Yaskawa INFORM job: aprem2TRJ3.JBI

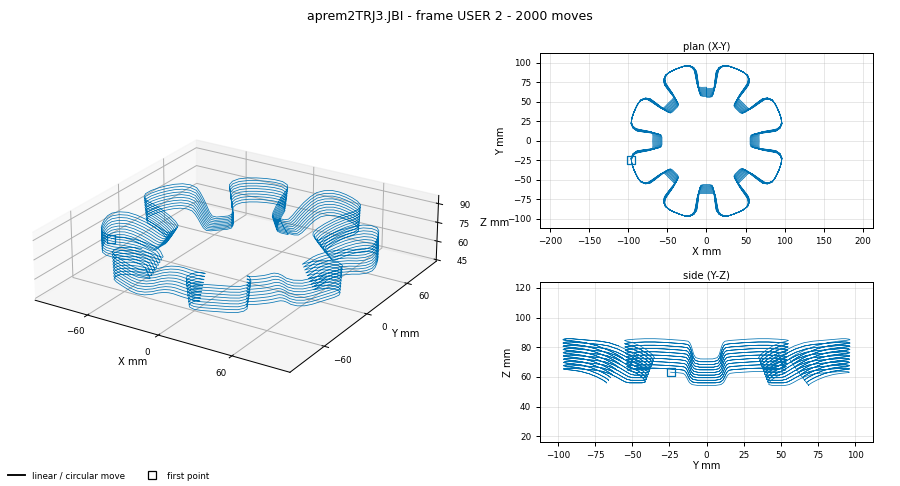
[picture p0: tool path of aprem2TRJ3.JBI in frame USER 2, 2000 of 2000 moves have a stored position in this frame; points joined in program order, loops and branches not executed]
/JOB
//NAME aprem2TRJ3
//POS
///NPOS 2000,0,2000,0,0,0
///USER 2
///TOOL 1
///POSTYPE USER
///RECTAN
///RCONF 1,0,0,0,0,0,0,0,0,0,0,0,0,0,0,0,0,0,0,0,0,0,0,0
C00000=-96.154,-24.159,63.210,179.7472,-2.4641,0.0000
C00001=-94.423,-19.246,62.877,177.2942,-4.1530,0.0000
C00002=-90.636,-15.942,62.469,172.7045,-3.4321,0.0000
C00003=-85.405,-14.621,61.698,172.2425,-1.7901,0.0000
C00004=-79.780,-13.569,60.151,174.0266,-1.3203,0.0000
C00005=-74.809,-12.586,58.158,176.9961,-0.7607,0.0000
C00006=-71.127,-11.507,56.252,-176.5790,1.2623,0.0000
C00007=-69.044,-9.699,54.888,-163.7838,26.3525,0.0000
C00008=-68.619,-6.200,54.350,-178.9508,38.3093,0.0000
C00009=-68.781,-2.945,54.326,177.7405,38.7530,0.0000
C00010=-68.843,0.000,54.342,179.9996,38.7765,0.0000
C00011=-68.781,2.945,54.326,-177.7401,38.7530,0.0000
C00012=-68.619,6.200,54.350,178.9482,38.3089,0.0000
C00013=-69.044,9.699,54.888,163.7840,26.3528,0.0000
C00014=-71.127,11.507,56.252,176.5790,1.2623,0.0000
C00015=-74.809,12.586,58.158,-176.9961,-0.7607,0.0000
C00016=-79.780,13.569,60.151,-174.0266,-1.3203,0.0000
C00017=-85.405,14.621,61.698,-172.2425,-1.7901,0.0000
C00018=-90.636,15.942,62.469,-172.7045,-3.4321,0.0000
C00019=-94.423,19.246,62.877,-177.2942,-4.1530,0.0000
C00020=-96.154,24.159,63.210,-179.7472,-2.4641,0.0000
C00021=-95.429,29.718,63.547,179.9546,-0.1514,0.0000
C00022=-93.512,35.416,63.770,179.9933,-0.0179,0.0000
C00023=-91.166,41.080,63.770,179.9921,-0.0174,0.0000
C00024=-88.493,46.465,63.547,179.9251,-0.1391,0.0000
C00025=-85.074,50.908,63.210,178.0786,-1.5643,0.0000
C00026=-80.376,53.158,62.877,175.1551,-1.0270,0.0000
C00027=-75.362,52.817,62.469,172.4279,2.7549,0.0000
C00028=-70.729,50.052,61.698,173.2462,4.2451,0.0000
C00029=-66.007,46.818,60.151,174.8410,3.3018,0.0000
C00030=-61.798,43.998,58.158,177.3380,1.5877,0.0000
C00031=-58.431,42.158,56.252,-176.6891,-1.5289,0.0000
C00032=-55.679,41.963,54.888,-150.9290,8.2296,0.0000
C00033=-52.905,44.137,54.350,-150.2488,28.6202,0.0000
C00034=-50.718,46.553,54.326,-151.6454,30.7727,0.0000
C00035=-48.679,48.679,54.342,-150.4014,29.5989,0.0000
C00036=-46.553,50.718,54.326,-149.2271,28.3544,0.0000
C00037=-44.137,52.905,54.350,-151.3816,29.7523,0.0000
C00038=-41.963,55.680,54.888,-171.7700,29.0711,0.0000
C00039=-42.158,58.431,56.252,178.4711,3.3109,0.0000
C00040=-43.998,61.798,58.158,-178.4123,-2.6620,0.0000
C00041=-46.818,66.007,60.151,-176.6982,-5.1590,0.0000
C00042=-50.052,70.729,61.698,-175.7549,-6.7538,0.0000
C00043=-52.817,75.362,62.469,-177.2451,-7.5721,0.0000
C00044=-53.158,80.376,62.877,178.9730,-4.8449,0.0000
C00045=-50.908,85.074,63.210,178.4357,-1.9214,0.0000
C00046=-46.465,88.493,63.547,179.8609,-0.0749,0.0000
C00047=-41.080,91.166,63.770,179.9826,-0.0079,0.0000
C00048=-35.416,93.512,63.770,179.9821,-0.0067,0.0000
C00049=-29.718,95.429,63.547,179.8486,-0.0454,0.0000
C00050=-24.159,96.154,63.210,177.5359,0.2528,0.0000
C00051=-19.246,94.423,62.877,175.8470,2.7058,0.0000
C00052=-15.942,90.636,62.469,176.5679,7.2955,0.0000
C00053=-14.621,85.405,61.698,178.2099,7.7575,0.0000
C00054=-13.569,79.780,60.151,178.6797,5.9734,0.0000
C00055=-12.586,74.809,58.158,179.2393,3.0039,0.0000
C00056=-11.507,71.127,56.252,-178.7377,-3.4210,0.0000
C00057=-9.699,69.044,54.888,-153.6472,-16.2160,0.0000
C00058=-6.200,68.619,54.350,-141.6911,-1.0518,0.0000
C00059=-2.945,68.781,54.326,-141.2470,2.2599,0.0000
C00060=0.000,68.843,54.342,-141.2235,-0.0004,0.0000
C00061=0.000,67.469,56.061,-141.5412,-0.0004,0.0000
C00062=2.820,67.413,56.044,-141.5636,-2.1988,0.0000
C00063=5.989,67.263,56.069,-142.0566,1.4090,0.0000
C00064=9.441,67.734,56.637,-154.9636,16.3668,0.0000
C00065=11.191,69.937,58.076,-179.1454,2.5065,0.0000
C00066=12.227,73.809,60.085,179.1943,-3.3815,0.0000
C00067=13.183,79.025,62.181,178.7261,-6.0865,0.0000
C00068=14.211,84.918,63.804,178.3204,-7.7435,0.0000
C00069=15.500,90.396,64.610,176.7328,-7.3164,0.0000
C00070=18.832,94.373,65.037,175.8897,-2.7823,0.0000
C00071=23.832,96.213,65.385,177.5484,-0.2740,0.0000
C00072=29.513,95.497,65.736,179.8479,0.0454,0.0000
C00073=35.347,93.539,65.969,179.9821,0.0067,0.0000
C00074=41.148,91.136,65.969,179.9826,0.0079,0.0000
C00075=46.658,88.395,65.736,179.8603,0.0754,0.0000
C00076=51.181,84.885,65.385,178.4595,1.9277,0.0000
C00077=53.416,80.048,65.037,179.0575,4.8686,0.0000
C00078=52.959,74.880,64.610,-177.1134,7.4719,0.0000
C00079=49.997,70.095,63.804,-175.6871,6.6669,0.0000
C00080=46.557,65.200,62.181,-176.5849,5.2066,0.0000
C00081=43.545,60.837,60.085,-178.1765,2.9610,0.0000
C00082=41.540,57.367,58.076,178.8310,-2.3765,0.0000
C00083=41.220,54.571,56.637,-173.0100,-28.2777,0.0000
C00084=43.327,51.796,56.069,-151.9006,-29.6278,0.0000
C00085=45.674,49.662,56.044,-149.5306,-28.1035,0.0000
C00086=47.708,47.708,56.061,-150.6800,-29.3196,0.0000
C00087=49.662,45.674,56.044,-151.8968,-30.4697,0.0000
C00088=51.797,43.327,56.069,-150.3712,-28.0975,0.0000
C00089=54.571,41.220,56.637,-151.7222,-6.9903,0.0000
C00090=57.367,41.540,58.076,-177.6235,1.1690,0.0000
C00091=60.837,43.545,60.085,177.0390,-1.8235,0.0000
C00092=65.200,46.557,62.181,174.7934,-3.4151,0.0000
C00093=70.095,49.997,63.804,173.3331,-4.3129,0.0000
C00094=74.880,52.959,64.610,172.5281,-2.8866,0.0000
C00095=80.048,53.416,65.037,175.1314,0.9425,0.0000
C00096=84.885,51.181,65.385,178.0723,1.5405,0.0000
C00097=88.395,46.658,65.736,179.9246,0.1397,0.0000
C00098=91.136,41.148,65.969,179.9921,0.0174,0.0000
C00099=93.539,35.347,65.969,179.9933,0.0179,0.0000
C00100=95.497,29.513,65.736,179.9546,0.1521,0.0000
C00101=96.213,23.832,65.385,-179.7260,2.4516,0.0000
C00102=94.373,18.832,65.037,-177.2177,4.1103,0.0000
C00103=90.396,15.500,64.610,-172.6836,3.2672,0.0000
C00104=84.918,14.211,63.804,-172.2565,1.6796,0.0000
C00105=79.025,13.183,62.181,-173.9135,1.2739,0.0000
C00106=73.809,12.227,60.085,-176.6185,0.8057,0.0000
C00107=69.937,11.191,58.076,177.4935,-0.8546,0.0000
C00108=67.734,9.441,56.637,163.6332,-25.0364,0.0000
C00109=67.263,5.989,56.069,178.5910,-37.9434,0.0000
C00110=67.413,2.820,56.044,-177.8012,-38.4364,0.0000
C00111=67.469,0.000,56.061,-179.9996,-38.4588,0.0000
C00112=67.413,-2.820,56.044,177.8008,-38.4364,0.0000
C00113=67.263,-5.989,56.069,-178.5883,-37.9429,0.0000
C00114=67.734,-9.441,56.637,-163.6333,-25.0366,0.0000
C00115=69.937,-11.191,58.076,-177.4935,-0.8546,0.0000
C00116=73.809,-12.227,60.085,176.6185,0.8057,0.0000
C00117=79.025,-13.183,62.181,173.9135,1.2739,0.0000
C00118=84.918,-14.211,63.804,172.2565,1.6796,0.0000
C00119=90.396,-15.500,64.610,172.6836,3.2672,0.0000
C00120=94.373,-18.832,65.037,177.2177,4.1103,0.0000
C00121=96.213,-23.832,65.385,179.7260,2.4516,0.0000
C00122=95.497,-29.513,65.736,-179.9546,0.1521,0.0000
C00123=93.539,-35.347,65.969,-179.9933,0.0179,0.0000
C00124=91.136,-41.148,65.969,-179.9921,0.0174,0.0000
C00125=88.395,-46.658,65.736,-179.9246,0.1397,0.0000
C00126=84.885,-51.181,65.385,-178.0723,1.5405,0.0000
C00127=80.048,-53.416,65.037,-175.1314,0.9425,0.0000
C00128=74.880,-52.959,64.610,-172.5281,-2.8866,0.0000
C00129=70.095,-49.997,63.804,-173.3331,-4.3129,0.0000
C00130=65.200,-46.557,62.181,-174.7934,-3.4151,0.0000
C00131=60.837,-43.545,60.085,-177.0390,-1.8235,0.0000
C00132=57.367,-41.540,58.076,177.6235,1.1690,0.0000
C00133=54.571,-41.220,56.637,151.7223,-6.9900,0.0000
C00134=51.796,-43.327,56.069,150.3722,-28.0994,0.0000
C00135=49.662,-45.674,56.044,151.8965,-30.4694,0.0000
C00136=47.708,-47.708,56.061,150.6804,-29.3200,0.0000
C00137=45.674,-49.662,56.044,149.5303,-28.1032,0.0000
C00138=43.327,-51.797,56.069,151.9025,-29.6288,0.0000
C00139=41.220,-54.571,56.637,173.0097,-28.2778,0.0000
C00140=41.540,-57.367,58.076,-178.8310,-2.3765,0.0000
C00141=43.545,-60.837,60.085,178.1765,2.9610,0.0000
C00142=46.557,-65.200,62.181,176.5849,5.2066,0.0000
C00143=49.997,-70.095,63.804,175.6871,6.6669,0.0000
C00144=52.959,-74.880,64.610,177.1134,7.4719,0.0000
C00145=53.416,-80.048,65.037,-179.0575,4.8686,0.0000
C00146=51.181,-84.885,65.385,-178.4595,1.9277,0.0000
C00147=46.658,-88.395,65.736,-179.8603,0.0754,0.0000
C00148=41.148,-91.136,65.969,-179.9826,0.0079,0.0000
C00149=35.347,-93.539,65.969,-179.9821,0.0067,0.0000
C00150=29.513,-95.497,65.736,-179.8479,0.0454,0.0000
C00151=23.832,-96.213,65.385,-177.5484,-0.2740,0.0000
C00152=18.832,-94.373,65.037,-175.8897,-2.7823,0.0000
C00153=15.500,-90.396,64.610,-176.7328,-7.3164,0.0000
C00154=14.211,-84.918,63.804,-178.3204,-7.7435,0.0000
C00155=13.183,-79.025,62.181,-178.7261,-6.0865,0.0000
C00156=12.227,-73.809,60.085,-179.1943,-3.3815,0.0000
C00157=11.191,-69.937,58.076,179.1454,2.5065,0.0000
C00158=9.441,-67.734,56.637,154.9636,16.3668,0.0000
C00159=5.989,-67.263,56.069,142.0566,1.4090,0.0000
C00160=2.820,-67.413,56.044,141.5636,-2.1988,0.0000
C00161=0.000,-67.469,56.061,141.5412,-0.0004,0.0000
C00162=0.000,-67.469,56.061,141.5412,-0.0004,0.0000
C00163=-2.820,-67.413,56.044,141.5636,2.1992,0.0000
C00164=-5.989,-67.263,56.069,142.0571,-1.4117,0.0000
C00165=-9.441,-67.734,56.637,154.9634,-16.3667,0.0000
C00166=-11.191,-69.937,58.076,179.1454,-2.5065,0.0000
C00167=-12.227,-73.809,60.085,-179.1943,3.3815,0.0000
C00168=-13.183,-79.025,62.181,-178.7261,6.0865,0.0000
C00169=-14.211,-84.918,63.804,-178.3204,7.7435,0.0000
C00170=-15.500,-90.396,64.610,-176.7328,7.3164,0.0000
C00171=-18.832,-94.373,65.037,-175.8897,2.7823,0.0000
C00172=-23.832,-96.213,65.385,-177.5484,0.2740,0.0000
C00173=-29.513,-95.497,65.736,-179.8479,-0.0454,0.0000
C00174=-35.347,-93.539,65.969,-179.9821,-0.0067,0.0000
C00175=-41.148,-91.136,65.969,-179.9826,-0.0079,0.0000
C00176=-46.658,-88.395,65.736,-179.8603,-0.0754,0.0000
C00177=-51.181,-84.885,65.385,-178.4595,-1.9277,0.0000
C00178=-53.416,-80.048,65.037,-179.0575,-4.8686,0.0000
C00179=-52.959,-74.880,64.610,177.1134,-7.4719,0.0000
C00180=-49.997,-70.095,63.804,175.6871,-6.6669,0.0000
C00181=-46.557,-65.200,62.181,176.5849,-5.2066,0.0000
C00182=-43.545,-60.837,60.085,178.1765,-2.9610,0.0000
C00183=-41.540,-57.367,58.076,-178.8310,2.3765,0.0000
C00184=-41.220,-54.571,56.637,173.0100,28.2777,0.0000
C00185=-43.327,-51.796,56.069,151.9006,29.6278,0.0000
C00186=-45.674,-49.662,56.044,149.5306,28.1035,0.0000
C00187=-47.708,-47.708,56.061,150.6800,29.3196,0.0000
C00188=-49.662,-45.674,56.044,151.8968,30.4697,0.0000
C00189=-51.797,-43.327,56.069,150.3712,28.0975,0.0000
C00190=-54.571,-41.220,56.637,151.7222,6.9903,0.0000
C00191=-57.367,-41.540,58.076,177.6235,-1.1690,0.0000
C00192=-60.837,-43.545,60.085,-177.0390,1.8235,0.0000
C00193=-65.200,-46.557,62.181,-174.7934,3.4151,0.0000
C00194=-70.095,-49.997,63.804,-173.3331,4.3129,0.0000
C00195=-74.880,-52.959,64.610,-172.5281,2.8866,0.0000
C00196=-80.048,-53.416,65.037,-175.1314,-0.9425,0.0000
C00197=-84.885,-51.181,65.385,-178.0723,-1.5405,0.0000
C00198=-88.395,-46.658,65.736,-179.9246,-0.1397,0.0000
C00199=-91.136,-41.148,65.969,-179.9921,-0.0174,0.0000
C00200=-93.539,-35.347,65.969,-179.9933,-0.0179,0.0000
C00201=-95.497,-29.513,65.736,-179.9546,-0.1521,0.0000
C00202=-96.213,-23.832,65.385,179.7260,-2.4516,0.0000
C00203=-94.373,-18.832,65.037,177.2177,-4.1103,0.0000
C00204=-90.396,-15.500,64.610,172.6836,-3.2672,0.0000
C00205=-84.918,-14.211,63.804,172.2565,-1.6796,0.0000
C00206=-79.025,-13.183,62.181,173.9135,-1.2739,0.0000
C00207=-73.809,-12.227,60.085,176.6185,-0.8057,0.0000
C00208=-69.937,-11.191,58.076,-177.4935,0.8546,0.0000
C00209=-67.734,-9.441,56.637,-163.6332,25.0364,0.0000
C00210=-67.263,-5.989,56.069,-178.5910,37.9434,0.0000
C00211=-67.413,-2.820,56.044,177.8012,38.4364,0.0000
C00212=-67.469,0.000,56.061,179.9996,38.4588,0.0000
C00213=-67.413,2.820,56.044,-177.8008,38.4364,0.0000
C00214=-67.263,5.989,56.069,178.5883,37.9429,0.0000
C00215=-67.734,9.441,56.637,163.6333,25.0366,0.0000
C00216=-69.937,11.191,58.076,177.4935,0.8546,0.0000
C00217=-73.809,12.227,60.085,-176.6185,-0.8057,0.0000
C00218=-79.025,13.183,62.181,-173.9135,-1.2739,0.0000
C00219=-84.918,14.211,63.804,-172.2565,-1.6796,0.0000
C00220=-90.396,15.500,64.610,-172.6836,-3.2672,0.0000
C00221=-94.373,18.832,65.037,-177.2177,-4.1103,0.0000
C00222=-96.213,23.832,65.385,-179.7260,-2.4516,0.0000
C00223=-95.497,29.513,65.736,179.9546,-0.1521,0.0000
C00224=-93.539,35.347,65.969,179.9933,-0.0179,0.0000
C00225=-91.136,41.148,65.969,179.9921,-0.0174,0.0000
C00226=-88.395,46.658,65.736,179.9246,-0.1397,0.0000
C00227=-84.885,51.181,65.385,178.0723,-1.5405,0.0000
C00228=-80.048,53.416,65.037,175.1314,-0.9425,0.0000
C00229=-74.880,52.959,64.610,172.5281,2.8866,0.0000
C00230=-70.095,49.997,63.804,173.3331,4.3129,0.0000
C00231=-65.200,46.557,62.181,174.7934,3.4151,0.0000
C00232=-60.837,43.545,60.085,177.0390,1.8235,0.0000
C00233=-57.367,41.540,58.076,-177.6235,-1.1690,0.0000
C00234=-54.571,41.220,56.637,-151.7223,6.9900,0.0000
C00235=-51.796,43.327,56.069,-150.3722,28.0994,0.0000
C00236=-49.662,45.674,56.044,-151.8965,30.4694,0.0000
C00237=-47.708,47.708,56.061,-150.6804,29.3200,0.0000
C00238=-45.674,49.662,56.044,-149.5303,28.1032,0.0000
C00239=-43.327,51.797,56.069,-151.9025,29.6288,0.0000
C00240=-41.220,54.571,56.637,-173.0097,28.2778,0.0000
C00241=-41.540,57.367,58.076,178.8310,2.3765,0.0000
C00242=-43.545,60.837,60.085,-178.1765,-2.9610,0.0000
C00243=-46.557,65.200,62.181,-176.5849,-5.2066,0.0000
C00244=-49.997,70.095,63.804,-175.6871,-6.6669,0.0000
C00245=-52.959,74.880,64.610,-177.1134,-7.4719,0.0000
C00246=-53.416,80.048,65.037,179.0575,-4.8686,0.0000
C00247=-51.181,84.885,65.385,178.4595,-1.9277,0.0000
C00248=-46.658,88.395,65.736,179.8603,-0.0754,0.0000
C00249=-41.148,91.136,65.969,179.9826,-0.0079,0.0000
C00250=-35.347,93.539,65.969,179.9821,-0.0067,0.0000
C00251=-29.513,95.497,65.736,179.8479,-0.0454,0.0000
C00252=-23.832,96.213,65.385,177.5484,0.2740,0.0000
C00253=-18.832,94.373,65.037,175.8897,2.7823,0.0000
C00254=-15.500,90.396,64.610,176.7328,7.3164,0.0000
C00255=-14.211,84.918,63.804,178.3204,7.7435,0.0000
C00256=-13.183,79.025,62.181,178.7261,6.0865,0.0000
C00257=-12.227,73.809,60.085,179.1943,3.3815,0.0000
C00258=-11.191,69.937,58.076,-179.1454,-2.5065,0.0000
C00259=-9.441,67.734,56.637,-154.9634,-16.3667,0.0000
C00260=-5.989,67.263,56.069,-142.0571,-1.4117,0.0000
C00261=-2.820,67.413,56.044,-141.5636,2.1992,0.0000
C00262=0.000,67.469,56.061,-141.5412,-0.0004,0.0000
C00263=0.000,66.107,57.788,-141.9405,-0.0005,0.0000
C00264=2.695,66.055,57.771,-141.9617,-2.1301,0.0000
C00265=5.779,65.917,57.797,-142.5088,1.7632,0.0000
C00266=9.185,66.436,58.394,-156.3340,16.3865,0.0000
C00267=10.880,68.762,59.909,-179.4729,1.6691,0.0000
C00268=11.874,72.826,62.021,179.1708,-3.6886,0.0000
C00269=12.805,78.288,64.219,178.7806,-6.1350,0.0000
C00270=13.814,84.445,65.915,178.4333,-7.6593,0.0000
C00271=15.073,90.163,66.756,176.9116,-7.2599,0.0000
C00272=18.432,94.325,67.200,175.9710,-2.8231,0.0000
C00273=23.517,96.271,67.561,177.5835,-0.2906,0.0000
C00274=29.315,95.562,67.927,179.8488,0.0450,0.0000
C00275=35.280,93.564,68.167,179.9823,0.0066,0.0000
C00276=41.213,91.107,68.167,179.9828,0.0078,0.0000
C00277=46.844,88.301,67.927,179.8613,0.0751,0.0000
C00278=51.445,84.703,67.561,178.4961,1.9145,0.0000
C00279=53.664,79.731,67.200,179.1443,4.8399,0.0000
C00280=53.097,74.413,66.756,-177.0274,7.3072,0.0000
C00281=49.944,69.479,65.915,-175.6680,6.5281,0.0000
C00282=46.303,64.413,64.219,-176.5119,5.2027,0.0000
C00283=43.100,59.892,62.021,-177.9754,3.1949,0.0000
C00284=40.929,56.315,59.909,179.1922,-1.5529,0.0000
C00285=40.483,53.472,58.394,-174.1779,-27.3765,0.0000
C00286=42.524,50.697,57.797,-152.4966,-29.4307,0.0000
C00287=44.802,48.614,57.771,-149.9071,-27.7853,0.0000
C00288=46.745,46.745,57.788,-151.0292,-28.9702,0.0000
C00289=48.613,44.802,57.771,-152.2149,-30.0932,0.0000
C00290=50.697,42.524,57.797,-150.5682,-27.5015,0.0000
C00291=53.472,40.483,58.395,-152.6235,-5.8223,0.0000
C00292=56.315,40.929,59.909,-178.4471,0.8078,0.0000
C00293=59.892,43.100,62.021,176.8051,-2.0246,0.0000
C00294=64.413,46.303,64.219,174.7973,-3.4881,0.0000
C00295=69.479,49.944,65.915,173.4719,-4.3320,0.0000
C00296=74.413,53.097,66.756,172.6928,-2.9726,0.0000
C00297=79.731,53.664,67.200,175.1601,0.8557,0.0000
C00298=84.703,51.445,67.561,178.0855,1.5039,0.0000
C00299=88.301,46.844,67.927,179.9249,0.1387,0.0000
C00300=91.107,41.213,68.167,179.9922,0.0172,0.0000
C00301=93.564,35.280,68.167,179.9934,0.0177,0.0000
C00302=95.562,29.315,67.927,179.9550,0.1512,0.0000
C00303=96.271,23.517,67.561,-179.7094,2.4165,0.0000
C00304=94.325,18.432,67.200,-177.1769,4.0290,0.0000
C00305=90.163,15.073,66.756,-172.7401,3.0884,0.0000
C00306=84.445,13.814,65.915,-172.3407,1.5667,0.0000
C00307=78.288,12.805,64.219,-173.8650,1.2194,0.0000
C00308=72.826,11.874,62.021,-176.3114,0.8292,0.0000
C00309=68.762,10.880,59.909,178.3309,-0.5271,0.0000
C00310=66.436,9.185,58.394,163.6135,-23.6660,0.0000
C00311=65.917,5.779,57.797,178.2368,-37.4912,0.0000
C00312=66.055,2.695,57.771,-177.8699,-38.0383,0.0000
C00313=66.107,0.000,57.788,-179.9995,-38.0595,0.0000
C00314=66.055,-2.695,57.771,177.8693,-38.0383,0.0000
C00315=65.917,-5.780,57.797,-178.2340,-37.4907,0.0000
C00316=66.436,-9.185,58.395,-163.6136,-23.6662,0.0000
C00317=68.762,-10.880,59.909,-178.3309,-0.5271,0.0000
C00318=72.826,-11.874,62.021,176.3114,0.8292,0.0000
C00319=78.288,-12.805,64.219,173.8650,1.2194,0.0000
C00320=84.445,-13.814,65.915,172.3407,1.5667,0.0000
C00321=90.163,-15.073,66.756,172.7401,3.0884,0.0000
C00322=94.325,-18.432,67.200,177.1769,4.0290,0.0000
C00323=96.271,-23.517,67.561,179.7094,2.4165,0.0000
C00324=95.562,-29.315,67.927,-179.9550,0.1512,0.0000
C00325=93.564,-35.280,68.167,-179.9934,0.0177,0.0000
C00326=91.107,-41.213,68.167,-179.9922,0.0172,0.0000
C00327=88.301,-46.844,67.927,-179.9249,0.1387,0.0000
C00328=84.703,-51.445,67.561,-178.0855,1.5039,0.0000
C00329=79.731,-53.664,67.200,-175.1601,0.8557,0.0000
C00330=74.413,-53.097,66.756,-172.6928,-2.9726,0.0000
C00331=69.479,-49.944,65.915,-173.4719,-4.3320,0.0000
C00332=64.413,-46.303,64.219,-174.7973,-3.4881,0.0000
C00333=59.892,-43.100,62.021,-176.8051,-2.0246,0.0000
C00334=56.315,-40.929,59.909,178.4471,0.8078,0.0000
C00335=53.472,-40.483,58.394,152.6235,-5.8221,0.0000
C00336=50.697,-42.524,57.797,150.5693,-27.5034,0.0000
C00337=48.614,-44.802,57.771,152.2147,-30.0929,0.0000
C00338=46.745,-46.745,57.788,151.0298,-28.9708,0.0000
C00339=44.802,-48.613,57.771,149.9068,-27.7851,0.0000
C00340=42.524,-50.697,57.797,152.4985,-29.4318,0.0000
C00341=40.483,-53.472,58.395,174.1777,-27.3765,0.0000
C00342=40.929,-56.315,59.909,-179.1922,-1.5529,0.0000
C00343=43.100,-59.892,62.021,177.9754,3.1949,0.0000
C00344=46.303,-64.413,64.219,176.5119,5.2027,0.0000
C00345=49.944,-69.479,65.915,175.6680,6.5281,0.0000
C00346=53.097,-74.413,66.756,177.0274,7.3072,0.0000
C00347=53.664,-79.731,67.200,-179.1443,4.8399,0.0000
C00348=51.445,-84.703,67.561,-178.4961,1.9145,0.0000
C00349=46.844,-88.301,67.927,-179.8613,0.0751,0.0000
C00350=41.213,-91.107,68.167,-179.9828,0.0078,0.0000
C00351=35.280,-93.564,68.167,-179.9823,0.0066,0.0000
C00352=29.315,-95.562,67.927,-179.8488,0.0450,0.0000
C00353=23.517,-96.271,67.561,-177.5835,-0.2906,0.0000
C00354=18.432,-94.325,67.200,-175.9710,-2.8231,0.0000
C00355=15.073,-90.163,66.756,-176.9116,-7.2599,0.0000
C00356=13.814,-84.445,65.915,-178.4333,-7.6593,0.0000
C00357=12.805,-78.288,64.219,-178.7806,-6.1350,0.0000
C00358=11.874,-72.826,62.021,-179.1708,-3.6886,0.0000
C00359=10.880,-68.762,59.909,179.4729,1.6691,0.0000
C00360=9.185,-66.436,58.394,156.3340,16.3865,0.0000
C00361=5.779,-65.917,57.797,142.5088,1.7632,0.0000
C00362=2.695,-66.055,57.771,141.9617,-2.1301,0.0000
C00363=0.000,-66.107,57.788,141.9405,-0.0005,0.0000
C00364=0.000,-66.107,57.788,141.9405,-0.0005,0.0000
C00365=-2.695,-66.055,57.771,141.9617,2.1307,0.0000
C00366=-5.780,-65.917,57.797,142.5093,-1.7660,0.0000
C00367=-9.185,-66.436,58.395,156.3338,-16.3864,0.0000
C00368=-10.880,-68.762,59.909,179.4729,-1.6691,0.0000
C00369=-11.874,-72.826,62.021,-179.1708,3.6886,0.0000
C00370=-12.805,-78.288,64.219,-178.7806,6.1350,0.0000
C00371=-13.814,-84.445,65.915,-178.4333,7.6593,0.0000
C00372=-15.073,-90.163,66.756,-176.9116,7.2599,0.0000
C00373=-18.432,-94.325,67.200,-175.9710,2.8231,0.0000
C00374=-23.517,-96.271,67.561,-177.5835,0.2906,0.0000
C00375=-29.315,-95.562,67.927,-179.8488,-0.0450,0.0000
C00376=-35.280,-93.564,68.167,-179.9823,-0.0066,0.0000
C00377=-41.213,-91.107,68.167,-179.9828,-0.0078,0.0000
C00378=-46.844,-88.301,67.927,-179.8613,-0.0751,0.0000
C00379=-51.445,-84.703,67.561,-178.4961,-1.9145,0.0000
C00380=-53.664,-79.731,67.200,-179.1443,-4.8399,0.0000
C00381=-53.097,-74.413,66.756,177.0274,-7.3072,0.0000
C00382=-49.944,-69.479,65.915,175.6680,-6.5281,0.0000
C00383=-46.303,-64.413,64.219,176.5119,-5.2027,0.0000
C00384=-43.100,-59.892,62.021,177.9754,-3.1949,0.0000
C00385=-40.929,-56.315,59.909,-179.1922,1.5529,0.0000
C00386=-40.483,-53.472,58.394,174.1779,27.3765,0.0000
C00387=-42.524,-50.697,57.797,152.4966,29.4307,0.0000
C00388=-44.802,-48.614,57.771,149.9071,27.7853,0.0000
C00389=-46.745,-46.745,57.788,151.0292,28.9702,0.0000
C00390=-48.613,-44.802,57.771,152.2149,30.0932,0.0000
C00391=-50.697,-42.524,57.797,150.5682,27.5015,0.0000
C00392=-53.472,-40.483,58.395,152.6235,5.8223,0.0000
C00393=-56.315,-40.929,59.909,178.4471,-0.8078,0.0000
C00394=-59.892,-43.100,62.021,-176.8051,2.0246,0.0000
C00395=-64.413,-46.303,64.219,-174.7973,3.4881,0.0000
C00396=-69.479,-49.944,65.915,-173.4719,4.3320,0.0000
C00397=-74.413,-53.097,66.756,-172.6928,2.9726,0.0000
C00398=-79.731,-53.664,67.200,-175.1601,-0.8557,0.0000
C00399=-84.703,-51.445,67.561,-178.0855,-1.5039,0.0000
C00400=-88.301,-46.844,67.927,-179.9249,-0.1387,0.0000
C00401=-91.107,-41.213,68.167,-179.9922,-0.0172,0.0000
C00402=-93.564,-35.280,68.167,-179.9934,-0.0177,0.0000
C00403=-95.562,-29.315,67.927,-179.9550,-0.1512,0.0000
C00404=-96.271,-23.517,67.561,179.7094,-2.4165,0.0000
C00405=-94.325,-18.432,67.200,177.1769,-4.0290,0.0000
C00406=-90.163,-15.073,66.756,172.7401,-3.0884,0.0000
C00407=-84.445,-13.814,65.915,172.3407,-1.5667,0.0000
C00408=-78.288,-12.805,64.219,173.8650,-1.2194,0.0000
C00409=-72.826,-11.874,62.021,176.3114,-0.8292,0.0000
C00410=-68.762,-10.880,59.909,-178.3309,0.5271,0.0000
C00411=-66.436,-9.185,58.394,-163.6135,23.6660,0.0000
C00412=-65.917,-5.779,57.797,-178.2368,37.4912,0.0000
C00413=-66.055,-2.695,57.771,177.8699,38.0383,0.0000
C00414=-66.107,0.000,57.788,179.9995,38.0595,0.0000
C00415=-66.055,2.695,57.771,-177.8693,38.0383,0.0000
C00416=-65.917,5.780,57.797,178.2340,37.4907,0.0000
C00417=-66.436,9.185,58.395,163.6136,23.6662,0.0000
C00418=-68.762,10.880,59.909,178.3309,0.5271,0.0000
C00419=-72.826,11.874,62.021,-176.3114,-0.8292,0.0000
C00420=-78.288,12.805,64.219,-173.8650,-1.2194,0.0000
C00421=-84.445,13.814,65.915,-172.3407,-1.5667,0.0000
C00422=-90.163,15.073,66.756,-172.7401,-3.0884,0.0000
C00423=-94.325,18.432,67.200,-177.1769,-4.0290,0.0000
C00424=-96.271,23.517,67.561,-179.7094,-2.4165,0.0000
C00425=-95.562,29.315,67.927,179.9550,-0.1512,0.0000
C00426=-93.564,35.280,68.167,179.9934,-0.0177,0.0000
C00427=-91.107,41.213,68.167,179.9922,-0.0172,0.0000
C00428=-88.301,46.844,67.927,179.9249,-0.1387,0.0000
C00429=-84.703,51.445,67.561,178.0855,-1.5039,0.0000
C00430=-79.731,53.664,67.200,175.1601,-0.8557,0.0000
C00431=-74.413,53.097,66.756,172.6928,2.9726,0.0000
C00432=-69.479,49.944,65.915,173.4719,4.3320,0.0000
C00433=-64.413,46.303,64.219,174.7973,3.4881,0.0000
C00434=-59.892,43.100,62.021,176.8051,2.0246,0.0000
C00435=-56.315,40.929,59.909,-178.4471,-0.8078,0.0000
C00436=-53.472,40.483,58.394,-152.6235,5.8221,0.0000
C00437=-50.697,42.524,57.797,-150.5693,27.5034,0.0000
C00438=-48.614,44.802,57.771,-152.2147,30.0929,0.0000
C00439=-46.745,46.745,57.788,-151.0298,28.9708,0.0000
C00440=-44.802,48.613,57.771,-149.9068,27.7851,0.0000
C00441=-42.524,50.697,57.797,-152.4985,29.4318,0.0000
C00442=-40.483,53.472,58.395,-174.1777,27.3765,0.0000
C00443=-40.929,56.315,59.909,179.1922,1.5529,0.0000
C00444=-43.100,59.892,62.021,-177.9754,-3.1949,0.0000
C00445=-46.303,64.413,64.219,-176.5119,-5.2027,0.0000
C00446=-49.944,69.479,65.915,-175.6680,-6.5281,0.0000
C00447=-53.097,74.413,66.756,-177.0274,-7.3072,0.0000
C00448=-53.664,79.731,67.200,179.1443,-4.8399,0.0000
C00449=-51.445,84.703,67.561,178.4961,-1.9145,0.0000
C00450=-46.844,88.301,67.927,179.8613,-0.0751,0.0000
C00451=-41.213,91.107,68.167,179.9828,-0.0078,0.0000
C00452=-35.280,93.564,68.167,179.9823,-0.0066,0.0000
C00453=-29.315,95.562,67.927,179.8488,-0.0450,0.0000
C00454=-23.517,96.271,67.561,177.5835,0.2906,0.0000
C00455=-18.432,94.325,67.200,175.9710,2.8231,0.0000
C00456=-15.073,90.163,66.756,176.9116,7.2599,0.0000
C00457=-13.814,84.445,65.915,178.4333,7.6593,0.0000
C00458=-12.805,78.288,64.219,178.7806,6.1350,0.0000
C00459=-11.874,72.826,62.021,179.1708,3.6886,0.0000
C00460=-10.880,68.762,59.909,-179.4729,-1.6691,0.0000
C00461=-9.185,66.436,58.395,-156.3338,-16.3864,0.0000
C00462=-5.780,65.917,57.797,-142.5093,-1.7660,0.0000
C00463=-2.695,66.055,57.771,-141.9617,2.1307,0.0000
C00464=0.000,66.107,57.788,-141.9405,-0.0005,0.0000
C00465=0.000,64.758,59.526,-142.4254,-0.0006,0.0000
C00466=2.572,64.710,59.508,-142.4454,-2.0536,0.0000
C00467=5.572,64.584,59.535,-143.0512,2.1076,0.0000
C00468=8.932,65.152,60.163,-157.7440,16.2795,0.0000
C00469=10.572,67.603,61.754,-179.7324,0.9128,0.0000
C00470=11.527,71.864,63.969,179.1649,-3.9269,0.0000
C00471=12.439,77.571,66.266,178.8415,-6.1204,0.0000
C00472=13.430,83.988,68.033,178.5474,-7.5065,0.0000
C00473=14.662,89.940,68.906,177.1014,-7.1283,0.0000
C00474=18.048,94.279,69.366,176.0893,-2.8270,0.0000
C00475=23.215,96.325,69.740,177.6414,-0.3022,0.0000
C00476=29.126,95.625,70.117,179.8514,0.0441,0.0000
C00477=35.216,93.589,70.366,179.9827,0.0065,0.0000
C00478=41.276,91.079,70.366,179.9832,0.0077,0.0000
C00479=47.022,88.212,70.117,179.8638,0.0739,0.0000
C00480=51.697,84.528,69.740,178.5453,1.8817,0.0000
C00481=53.903,79.427,69.366,179.2311,4.7592,0.0000
C00482=53.229,73.964,68.906,-176.9875,7.0817,0.0000
C00483=49.892,68.885,68.033,-175.6970,6.3398,0.0000
C00484=46.056,63.647,66.266,-176.4794,5.1497,0.0000
C00485=42.664,58.966,63.969,-177.8105,3.3678,0.0000
C00486=40.327,55.279,61.754,179.5437,-0.8347,0.0000
C00487=39.754,52.385,60.163,-175.2625,-26.3754,0.0000
C00488=41.728,49.608,59.535,-153.1683,-29.1561,0.0000
C00489=43.938,47.576,59.508,-150.3598,-27.3976,0.0000
C00490=45.791,45.791,59.526,-151.4514,-28.5479,0.0000
C00491=47.575,43.938,59.508,-152.6027,-29.6406,0.0000
C00492=49.608,41.728,59.535,-150.8429,-26.8297,0.0000
C00493=52.385,39.754,60.163,-153.6246,-4.7376,0.0000
C00494=55.279,40.327,61.754,-179.1653,0.4563,0.0000
C00495=58.966,42.664,63.969,176.6322,-2.1895,0.0000
C00496=63.647,46.056,66.266,174.8503,-3.5206,0.0000
C00497=68.885,49.892,68.033,173.6602,-4.3030,0.0000
C00498=73.964,53.229,68.906,172.9183,-3.0125,0.0000
C00499=79.427,53.903,69.366,175.2408,0.7689,0.0000
C00500=84.528,51.697,69.740,178.1183,1.4547,0.0000
C00501=88.212,47.022,70.117,179.9261,0.1362,0.0000
C00502=91.079,41.276,70.366,179.9923,0.0168,0.0000
C00503=93.589,35.216,70.366,179.9935,0.0173,0.0000
C00504=95.625,29.126,70.117,179.9559,0.1486,0.0000
C00505=96.325,23.215,69.740,-179.6978,2.3586,0.0000
C00506=94.279,18.048,69.366,-177.1730,3.9107,0.0000
C00507=89.940,14.662,68.906,-172.8717,2.8986,0.0000
C00508=83.988,13.430,68.033,-172.4935,1.4526,0.0000
C00509=77.571,12.439,66.266,-173.8796,1.1585,0.0000
C00510=71.864,11.527,63.969,-176.0731,0.8351,0.0000
C00511=67.603,10.572,61.754,179.0872,-0.2676,0.0000
C00512=65.152,8.932,60.163,163.7205,-22.2560,0.0000
C00513=64.584,5.572,59.535,177.8924,-36.9488,0.0000
C00514=64.710,2.572,59.508,-177.9464,-37.5546,0.0000
C00515=64.758,0.000,59.526,-179.9994,-37.5746,0.0000
C00516=64.710,-2.572,59.508,177.9458,-37.5546,0.0000
C00517=64.584,-5.572,59.535,-177.8896,-36.9483,0.0000
C00518=65.152,-8.932,60.163,-163.7206,-22.2560,0.0000
C00519=67.603,-10.572,61.754,-179.0872,-0.2676,0.0000
C00520=71.864,-11.527,63.969,176.0731,0.8351,0.0000
C00521=77.571,-12.439,66.266,173.8796,1.1585,0.0000
C00522=83.988,-13.430,68.033,172.4935,1.4526,0.0000
C00523=89.940,-14.662,68.906,172.8717,2.8986,0.0000
C00524=94.279,-18.048,69.366,177.1730,3.9107,0.0000
C00525=96.325,-23.215,69.740,179.6978,2.3586,0.0000
C00526=95.625,-29.126,70.117,-179.9559,0.1486,0.0000
C00527=93.589,-35.216,70.366,-179.9935,0.0173,0.0000
C00528=91.079,-41.276,70.366,-179.9923,0.0168,0.0000
C00529=88.212,-47.022,70.117,-179.9261,0.1362,0.0000
C00530=84.528,-51.697,69.740,-178.1183,1.4547,0.0000
C00531=79.427,-53.903,69.366,-175.2408,0.7689,0.0000
C00532=73.964,-53.229,68.906,-172.9183,-3.0125,0.0000
C00533=68.885,-49.892,68.033,-173.6602,-4.3030,0.0000
C00534=63.647,-46.056,66.266,-174.8503,-3.5206,0.0000
C00535=58.966,-42.664,63.969,-176.6322,-2.1895,0.0000
C00536=55.279,-40.327,61.754,179.1653,0.4563,0.0000
C00537=52.385,-39.754,60.163,153.6246,-4.7375,0.0000
C00538=49.608,-41.728,59.535,150.8439,-26.8317,0.0000
C00539=47.576,-43.938,59.508,152.6024,-29.6402,0.0000
C00540=45.791,-45.791,59.526,151.4521,-28.5486,0.0000
C00541=43.938,-47.575,59.508,150.3594,-27.3973,0.0000
C00542=41.728,-49.608,59.535,153.1703,-29.1571,0.0000
C00543=39.754,-52.385,60.163,175.2624,-26.3754,0.0000
C00544=40.327,-55.279,61.754,-179.5437,-0.8347,0.0000
C00545=42.664,-58.966,63.969,177.8105,3.3678,0.0000
C00546=46.056,-63.647,66.266,176.4794,5.1497,0.0000
C00547=49.892,-68.885,68.033,175.6970,6.3398,0.0000
C00548=53.229,-73.964,68.906,176.9875,7.0817,0.0000
C00549=53.903,-79.427,69.366,-179.2311,4.7592,0.0000
C00550=51.697,-84.528,69.740,-178.5453,1.8817,0.0000
C00551=47.022,-88.212,70.117,-179.8638,0.0739,0.0000
C00552=41.276,-91.079,70.366,-179.9832,0.0077,0.0000
C00553=35.216,-93.589,70.366,-179.9827,0.0065,0.0000
C00554=29.126,-95.625,70.117,-179.8514,0.0441,0.0000
C00555=23.215,-96.325,69.740,-177.6414,-0.3022,0.0000
C00556=18.048,-94.279,69.366,-176.0893,-2.8270,0.0000
C00557=14.662,-89.940,68.906,-177.1014,-7.1283,0.0000
C00558=13.430,-83.988,68.033,-178.5474,-7.5065,0.0000
C00559=12.439,-77.571,66.266,-178.8415,-6.1204,0.0000
C00560=11.527,-71.864,63.969,-179.1649,-3.9269,0.0000
C00561=10.572,-67.603,61.754,179.7324,0.9128,0.0000
C00562=8.932,-65.152,60.163,157.7440,16.2795,0.0000
C00563=5.572,-64.584,59.535,143.0512,2.1076,0.0000
C00564=2.572,-64.710,59.508,142.4454,-2.0536,0.0000
C00565=0.000,-64.758,59.526,142.4254,-0.0006,0.0000
C00566=0.000,-64.758,59.526,142.4254,-0.0006,0.0000
C00567=-2.572,-64.710,59.508,142.4454,2.0542,0.0000
C00568=-5.572,-64.584,59.535,143.0517,-2.1104,0.0000
C00569=-8.932,-65.152,60.163,157.7440,-16.2794,0.0000
C00570=-10.572,-67.603,61.754,179.7324,-0.9128,0.0000
C00571=-11.527,-71.864,63.969,-179.1649,3.9269,0.0000
C00572=-12.439,-77.571,66.266,-178.8415,6.1204,0.0000
C00573=-13.430,-83.988,68.033,-178.5474,7.5065,0.0000
C00574=-14.662,-89.940,68.906,-177.1014,7.1283,0.0000
C00575=-18.048,-94.279,69.366,-176.0893,2.8270,0.0000
C00576=-23.215,-96.325,69.740,-177.6414,0.3022,0.0000
C00577=-29.126,-95.625,70.117,-179.8514,-0.0441,0.0000
C00578=-35.216,-93.589,70.366,-179.9827,-0.0065,0.0000
C00579=-41.276,-91.079,70.366,-179.9832,-0.0077,0.0000
C00580=-47.022,-88.212,70.117,-179.8638,-0.0739,0.0000
C00581=-51.697,-84.528,69.740,-178.5453,-1.8817,0.0000
C00582=-53.903,-79.427,69.366,-179.2311,-4.7592,0.0000
C00583=-53.229,-73.964,68.906,176.9875,-7.0817,0.0000
C00584=-49.892,-68.885,68.033,175.6970,-6.3398,0.0000
C00585=-46.056,-63.647,66.266,176.4794,-5.1497,0.0000
C00586=-42.664,-58.966,63.969,177.8105,-3.3678,0.0000
C00587=-40.327,-55.279,61.754,-179.5437,0.8347,0.0000
C00588=-39.754,-52.385,60.163,175.2625,26.3754,0.0000
C00589=-41.728,-49.608,59.535,153.1683,29.1561,0.0000
C00590=-43.938,-47.576,59.508,150.3598,27.3976,0.0000
C00591=-45.791,-45.791,59.526,151.4514,28.5479,0.0000
C00592=-47.575,-43.938,59.508,152.6027,29.6406,0.0000
C00593=-49.608,-41.728,59.535,150.8429,26.8297,0.0000
C00594=-52.385,-39.754,60.163,153.6246,4.7376,0.0000
C00595=-55.279,-40.327,61.754,179.1653,-0.4563,0.0000
C00596=-58.966,-42.664,63.969,-176.6322,2.1895,0.0000
C00597=-63.647,-46.056,66.266,-174.8503,3.5206,0.0000
C00598=-68.885,-49.892,68.033,-173.6602,4.3030,0.0000
C00599=-73.964,-53.229,68.906,-172.9183,3.0125,0.0000
C00600=-79.427,-53.903,69.366,-175.2408,-0.7689,0.0000
C00601=-84.528,-51.697,69.740,-178.1183,-1.4547,0.0000
C00602=-88.212,-47.022,70.117,-179.9261,-0.1362,0.0000
C00603=-91.079,-41.276,70.366,-179.9923,-0.0168,0.0000
C00604=-93.589,-35.216,70.366,-179.9935,-0.0173,0.0000
C00605=-95.625,-29.126,70.117,-179.9559,-0.1486,0.0000
C00606=-96.325,-23.215,69.740,179.6978,-2.3586,0.0000
C00607=-94.279,-18.048,69.366,177.1730,-3.9107,0.0000
C00608=-89.940,-14.662,68.906,172.8717,-2.8986,0.0000
C00609=-83.988,-13.430,68.033,172.4935,-1.4526,0.0000
C00610=-77.571,-12.439,66.266,173.8796,-1.1585,0.0000
C00611=-71.864,-11.527,63.969,176.0731,-0.8351,0.0000
C00612=-67.603,-10.572,61.754,-179.0872,0.2676,0.0000
C00613=-65.152,-8.932,60.163,-163.7205,22.2560,0.0000
C00614=-64.584,-5.572,59.535,-177.8924,36.9488,0.0000
C00615=-64.710,-2.572,59.508,177.9464,37.5546,0.0000
C00616=-64.758,0.000,59.526,179.9994,37.5746,0.0000
C00617=-64.710,2.572,59.508,-177.9458,37.5546,0.0000
C00618=-64.584,5.572,59.535,177.8896,36.9483,0.0000
C00619=-65.152,8.932,60.163,163.7206,22.2560,0.0000
C00620=-67.603,10.572,61.754,179.0872,0.2676,0.0000
C00621=-71.864,11.527,63.969,-176.0731,-0.8351,0.0000
C00622=-77.571,12.439,66.266,-173.8796,-1.1585,0.0000
C00623=-83.988,13.430,68.033,-172.4935,-1.4526,0.0000
C00624=-89.940,14.662,68.906,-172.8717,-2.8986,0.0000
C00625=-94.279,18.048,69.366,-177.1730,-3.9107,0.0000
C00626=-96.325,23.215,69.740,-179.6978,-2.3586,0.0000
C00627=-95.625,29.126,70.117,179.9559,-0.1486,0.0000
C00628=-93.589,35.216,70.366,179.9935,-0.0173,0.0000
C00629=-91.079,41.276,70.366,179.9923,-0.0168,0.0000
C00630=-88.212,47.022,70.117,179.9261,-0.1362,0.0000
C00631=-84.528,51.697,69.740,178.1183,-1.4547,0.0000
C00632=-79.427,53.903,69.366,175.2408,-0.7689,0.0000
C00633=-73.964,53.229,68.906,172.9183,3.0125,0.0000
C00634=-68.885,49.892,68.033,173.6602,4.3030,0.0000
C00635=-63.647,46.056,66.266,174.8503,3.5206,0.0000
C00636=-58.966,42.664,63.969,176.6322,2.1895,0.0000
C00637=-55.279,40.327,61.754,-179.1653,-0.4563,0.0000
C00638=-52.385,39.754,60.163,-153.6246,4.7375,0.0000
C00639=-49.608,41.728,59.535,-150.8439,26.8317,0.0000
C00640=-47.576,43.938,59.508,-152.6024,29.6402,0.0000
C00641=-45.791,45.791,59.526,-151.4521,28.5486,0.0000
C00642=-43.938,47.575,59.508,-150.3594,27.3973,0.0000
C00643=-41.728,49.608,59.535,-153.1703,29.1571,0.0000
C00644=-39.754,52.385,60.163,-175.2624,26.3754,0.0000
C00645=-40.327,55.279,61.754,179.5437,0.8347,0.0000
C00646=-42.664,58.966,63.969,-177.8105,-3.3678,0.0000
C00647=-46.056,63.647,66.266,-176.4794,-5.1497,0.0000
C00648=-49.892,68.885,68.033,-175.6970,-6.3398,0.0000
C00649=-53.229,73.964,68.906,-176.9875,-7.0817,0.0000
C00650=-53.903,79.427,69.366,179.2311,-4.7592,0.0000
C00651=-51.697,84.528,69.740,178.5453,-1.8817,0.0000
C00652=-47.022,88.212,70.117,179.8638,-0.0739,0.0000
C00653=-41.276,91.079,70.366,179.9832,-0.0077,0.0000
C00654=-35.216,93.589,70.366,179.9827,-0.0065,0.0000
C00655=-29.126,95.625,70.117,179.8514,-0.0441,0.0000
C00656=-23.215,96.325,69.740,177.6414,0.3022,0.0000
C00657=-18.048,94.279,69.366,176.0893,2.8270,0.0000
C00658=-14.662,89.940,68.906,177.1014,7.1283,0.0000
C00659=-13.430,83.988,68.033,178.5474,7.5065,0.0000
C00660=-12.439,77.571,66.266,178.8415,6.1204,0.0000
C00661=-11.527,71.864,63.969,179.1649,3.9269,0.0000
C00662=-10.572,67.603,61.754,-179.7324,-0.9128,0.0000
C00663=-8.932,65.152,60.163,-157.7440,-16.2794,0.0000
C00664=-5.572,64.584,59.535,-143.0517,-2.1104,0.0000
C00665=-2.572,64.710,59.508,-142.4454,2.0542,0.0000
C00666=0.000,64.758,59.526,-142.4254,-0.0006,0.0000
C00667=0.000,63.425,61.276,-143.0012,-0.0007,0.0000
C00668=2.450,63.381,61.257,-143.0199,-1.9693,0.0000
C00669=5.367,63.268,61.285,-143.6888,2.4374,0.0000
C00670=8.682,63.886,61.945,-159.1792,16.0512,0.0000
C00671=10.270,66.465,63.612,-179.9346,0.2399,0.0000
C00672=11.189,70.924,65.929,179.1735,-4.0983,0.0000
C00673=12.084,76.878,68.324,178.9074,-6.0442,0.0000
C00674=13.063,83.550,70.157,178.6617,-7.2870,0.0000
C00675=14.270,89.726,71.060,177.3000,-6.9235,0.0000
C00676=17.683,94.235,71.535,176.2430,-2.7934,0.0000
C00677=22.929,96.378,71.920,177.7221,-0.3083,0.0000
C00678=28.946,95.684,72.309,179.8557,0.0426,0.0000
C00679=35.156,93.612,72.565,179.9833,0.0062,0.0000
C00680=41.335,91.053,72.565,179.9837,0.0074,0.0000
C00681=47.191,88.127,72.309,179.8678,0.0719,0.0000
C00682=51.936,84.362,71.920,178.6067,1.8290,0.0000
C00683=54.130,79.138,71.535,179.3164,4.6272,0.0000
C00684=53.356,73.536,71.060,-176.9938,6.7981,0.0000
C00685=49.842,68.316,70.157,-175.7735,6.1039,0.0000
C00686=45.816,62.906,68.324,-176.4873,5.0494,0.0000
C00687=42.239,58.063,65.929,-177.6829,3.4831,0.0000
C00688=39.736,54.260,63.612,179.8766,-0.2159,0.0000
C00689=39.035,51.313,61.945,-176.2551,-25.2833,0.0000
C00690=40.942,48.532,61.285,-153.9166,-28.7991,0.0000
C00691=43.085,46.550,61.257,-150.8922,-26.9372,0.0000
C00692=44.848,44.848,61.276,-151.9501,-28.0492,0.0000
C00693=46.550,43.085,61.257,-153.0632,-29.1083,0.0000
C00694=48.532,40.942,61.285,-151.1999,-26.0813,0.0000
C00695=51.313,39.035,61.945,-154.7168,-3.7449,0.0000
C00696=54.260,39.736,63.612,-179.7841,0.1234,0.0000
C00697=58.063,42.239,65.929,176.5169,-2.3171,0.0000
C00698=62.906,45.816,68.324,174.9506,-3.5127,0.0000
C00699=68.316,49.842,70.157,173.8961,-4.2265,0.0000
C00700=73.536,53.356,71.060,173.2019,-3.0062,0.0000
C00701=79.138,54.130,71.535,175.3728,0.6836,0.0000
C00702=84.362,51.936,71.920,178.1710,1.3933,0.0000
C00703=88.127,47.191,72.309,179.9281,0.1322,0.0000
C00704=91.053,41.335,72.565,179.9926,0.0163,0.0000
C00705=93.612,35.156,72.565,179.9938,0.0167,0.0000
C00706=95.684,28.946,72.309,179.9574,0.1443,0.0000
C00707=96.378,22.929,71.920,-179.6917,2.2779,0.0000
C00708=94.235,17.683,71.535,-177.2066,3.7570,0.0000
C00709=89.726,14.270,71.060,-173.0765,2.7000,0.0000
C00710=83.550,13.063,70.157,-172.7130,1.3383,0.0000
C00711=76.878,12.084,68.324,-173.9558,1.0926,0.0000
C00712=70.924,11.189,65.929,-175.9017,0.8265,0.0000
C00713=66.465,10.270,63.612,179.7601,-0.0654,0.0000
C00714=63.886,8.682,61.945,163.9488,-20.8208,0.0000
C00715=63.268,5.367,61.285,177.5626,-36.3112,0.0000
C00716=63.381,2.450,61.257,-178.0307,-36.9801,0.0000
C00717=63.425,0.000,61.276,-179.9993,-36.9988,0.0000
C00718=63.381,-2.450,61.257,178.0299,-36.9802,0.0000
C00719=63.268,-5.367,61.285,-177.5598,-36.3106,0.0000
C00720=63.886,-8.682,61.945,-163.9488,-20.8207,0.0000
C00721=66.465,-10.270,63.612,-179.7601,-0.0654,0.0000
C00722=70.924,-11.189,65.929,175.9017,0.8265,0.0000
C00723=76.878,-12.084,68.324,173.9558,1.0926,0.0000
C00724=83.550,-13.063,70.157,172.7130,1.3383,0.0000
C00725=89.726,-14.270,71.060,173.0765,2.7000,0.0000
C00726=94.235,-17.683,71.535,177.2066,3.7570,0.0000
C00727=96.378,-22.929,71.920,179.6917,2.2779,0.0000
C00728=95.684,-28.946,72.309,-179.9574,0.1443,0.0000
C00729=93.612,-35.156,72.565,-179.9938,0.0167,0.0000
C00730=91.053,-41.335,72.565,-179.9926,0.0163,0.0000
C00731=88.127,-47.191,72.309,-179.9281,0.1322,0.0000
C00732=84.362,-51.936,71.920,-178.1710,1.3933,0.0000
C00733=79.138,-54.130,71.535,-175.3728,0.6836,0.0000
C00734=73.536,-53.356,71.060,-173.2019,-3.0062,0.0000
C00735=68.316,-49.842,70.157,-173.8961,-4.2265,0.0000
C00736=62.906,-45.816,68.324,-174.9506,-3.5127,0.0000
C00737=58.063,-42.239,65.929,-176.5169,-2.3171,0.0000
C00738=54.260,-39.736,63.612,179.7841,0.1234,0.0000
C00739=51.313,-39.035,61.945,154.7167,-3.7449,0.0000
C00740=48.532,-40.942,61.285,151.2009,-26.0834,0.0000
C00741=46.550,-43.085,61.257,153.0628,-29.1078,0.0000
C00742=44.848,-44.848,61.276,151.9508,-28.0499,0.0000
C00743=43.085,-46.550,61.257,150.8917,-26.9368,0.0000
C00744=40.942,-48.532,61.285,153.9187,-28.8001,0.0000
C00745=39.035,-51.313,61.945,176.2551,-25.2832,0.0000
C00746=39.736,-54.260,63.612,-179.8766,-0.2159,0.0000
C00747=42.239,-58.063,65.929,177.6829,3.4831,0.0000
C00748=45.816,-62.906,68.324,176.4873,5.0494,0.0000
C00749=49.842,-68.316,70.157,175.7735,6.1039,0.0000
C00750=53.356,-73.536,71.060,176.9938,6.7981,0.0000
C00751=54.130,-79.138,71.535,-179.3164,4.6272,0.0000
C00752=51.936,-84.362,71.920,-178.6067,1.8290,0.0000
C00753=47.191,-88.127,72.309,-179.8678,0.0719,0.0000
C00754=41.335,-91.053,72.565,-179.9837,0.0074,0.0000
C00755=35.156,-93.612,72.565,-179.9833,0.0062,0.0000
C00756=28.946,-95.684,72.309,-179.8557,0.0426,0.0000
C00757=22.929,-96.378,71.920,-177.7221,-0.3083,0.0000
C00758=17.683,-94.235,71.535,-176.2430,-2.7934,0.0000
C00759=14.270,-89.726,71.060,-177.3000,-6.9235,0.0000
C00760=13.063,-83.550,70.157,-178.6617,-7.2870,0.0000
C00761=12.084,-76.878,68.324,-178.9074,-6.0442,0.0000
C00762=11.189,-70.924,65.929,-179.1735,-4.0983,0.0000
C00763=10.270,-66.465,63.612,179.9346,0.2399,0.0000
C00764=8.682,-63.886,61.945,159.1792,16.0512,0.0000
C00765=5.367,-63.268,61.285,143.6888,2.4374,0.0000
C00766=2.450,-63.381,61.257,143.0199,-1.9693,0.0000
C00767=0.000,-63.425,61.276,143.0012,-0.0007,0.0000
C00768=0.000,-63.425,61.276,143.0012,-0.0007,0.0000
C00769=-2.450,-63.381,61.257,143.0198,1.9701,0.0000
C00770=-5.367,-63.268,61.285,143.6894,-2.4402,0.0000
C00771=-8.682,-63.886,61.945,159.1793,-16.0512,0.0000
C00772=-10.270,-66.465,63.612,179.9346,-0.2399,0.0000
C00773=-11.189,-70.924,65.929,-179.1735,4.0983,0.0000
C00774=-12.084,-76.878,68.324,-178.9074,6.0442,0.0000
C00775=-13.063,-83.550,70.157,-178.6617,7.2870,0.0000
C00776=-14.270,-89.726,71.060,-177.3000,6.9235,0.0000
C00777=-17.683,-94.235,71.535,-176.2430,2.7934,0.0000
C00778=-22.929,-96.378,71.920,-177.7221,0.3083,0.0000
C00779=-28.946,-95.684,72.309,-179.8557,-0.0426,0.0000
C00780=-35.156,-93.612,72.565,-179.9833,-0.0062,0.0000
C00781=-41.335,-91.053,72.565,-179.9837,-0.0074,0.0000
C00782=-47.191,-88.127,72.309,-179.8678,-0.0719,0.0000
C00783=-51.936,-84.362,71.920,-178.6067,-1.8290,0.0000
C00784=-54.130,-79.138,71.535,-179.3164,-4.6272,0.0000
C00785=-53.356,-73.536,71.060,176.9938,-6.7981,0.0000
C00786=-49.842,-68.316,70.157,175.7735,-6.1039,0.0000
C00787=-45.816,-62.906,68.324,176.4873,-5.0494,0.0000
C00788=-42.239,-58.063,65.929,177.6829,-3.4831,0.0000
C00789=-39.736,-54.260,63.612,-179.8766,0.2159,0.0000
C00790=-39.035,-51.313,61.945,176.2551,25.2833,0.0000
C00791=-40.942,-48.532,61.285,153.9166,28.7991,0.0000
C00792=-43.085,-46.550,61.257,150.8922,26.9372,0.0000
C00793=-44.848,-44.848,61.276,151.9501,28.0492,0.0000
C00794=-46.550,-43.085,61.257,153.0632,29.1083,0.0000
C00795=-48.532,-40.942,61.285,151.1999,26.0813,0.0000
C00796=-51.313,-39.035,61.945,154.7168,3.7449,0.0000
C00797=-54.260,-39.736,63.612,179.7841,-0.1234,0.0000
C00798=-58.063,-42.239,65.929,-176.5169,2.3171,0.0000
C00799=-62.906,-45.816,68.324,-174.9506,3.5127,0.0000
C00800=-68.316,-49.842,70.157,-173.8961,4.2265,0.0000
C00801=-73.536,-53.356,71.060,-173.2019,3.0062,0.0000
C00802=-79.138,-54.130,71.535,-175.3728,-0.6836,0.0000
C00803=-84.362,-51.936,71.920,-178.1710,-1.3933,0.0000
C00804=-88.127,-47.191,72.309,-179.9281,-0.1322,0.0000
C00805=-91.053,-41.335,72.565,-179.9926,-0.0163,0.0000
C00806=-93.612,-35.156,72.565,-179.9938,-0.0167,0.0000
C00807=-95.684,-28.946,72.309,-179.9574,-0.1443,0.0000
C00808=-96.378,-22.929,71.920,179.6917,-2.2779,0.0000
C00809=-94.235,-17.683,71.535,177.2066,-3.7570,0.0000
C00810=-89.726,-14.270,71.060,173.0765,-2.7000,0.0000
C00811=-83.550,-13.063,70.157,172.7130,-1.3383,0.0000
C00812=-76.878,-12.084,68.324,173.9558,-1.0926,0.0000
C00813=-70.924,-11.189,65.929,175.9017,-0.8265,0.0000
C00814=-66.465,-10.270,63.612,-179.7601,0.0654,0.0000
C00815=-63.886,-8.682,61.945,-163.9488,20.8208,0.0000
C00816=-63.268,-5.367,61.285,-177.5626,36.3112,0.0000
C00817=-63.381,-2.450,61.257,178.0307,36.9801,0.0000
C00818=-63.425,0.000,61.276,179.9993,36.9988,0.0000
C00819=-63.381,2.450,61.257,-178.0299,36.9802,0.0000
C00820=-63.268,5.367,61.285,177.5598,36.3106,0.0000
C00821=-63.886,8.682,61.945,163.9488,20.8207,0.0000
C00822=-66.465,10.270,63.612,179.7601,0.0654,0.0000
C00823=-70.924,11.189,65.929,-175.9017,-0.8265,0.0000
C00824=-76.878,12.084,68.324,-173.9558,-1.0926,0.0000
C00825=-83.550,13.063,70.157,-172.7130,-1.3383,0.0000
C00826=-89.726,14.270,71.060,-173.0765,-2.7000,0.0000
C00827=-94.235,17.683,71.535,-177.2066,-3.7570,0.0000
C00828=-96.378,22.929,71.920,-179.6917,-2.2779,0.0000
C00829=-95.684,28.946,72.309,179.9574,-0.1443,0.0000
C00830=-93.612,35.156,72.565,179.9938,-0.0167,0.0000
C00831=-91.053,41.335,72.565,179.9926,-0.0163,0.0000
C00832=-88.127,47.191,72.309,179.9281,-0.1322,0.0000
C00833=-84.362,51.936,71.920,178.1710,-1.3933,0.0000
C00834=-79.138,54.130,71.535,175.3728,-0.6836,0.0000
C00835=-73.536,53.356,71.060,173.2019,3.0062,0.0000
C00836=-68.316,49.842,70.157,173.8961,4.2265,0.0000
C00837=-62.906,45.816,68.324,174.9506,3.5127,0.0000
C00838=-58.063,42.239,65.929,176.5169,2.3171,0.0000
C00839=-54.260,39.736,63.612,-179.7841,-0.1234,0.0000
C00840=-51.313,39.035,61.945,-154.7167,3.7449,0.0000
C00841=-48.532,40.942,61.285,-151.2009,26.0834,0.0000
C00842=-46.550,43.085,61.257,-153.0628,29.1078,0.0000
C00843=-44.848,44.848,61.276,-151.9508,28.0499,0.0000
C00844=-43.085,46.550,61.257,-150.8917,26.9368,0.0000
C00845=-40.942,48.532,61.285,-153.9187,28.8001,0.0000
C00846=-39.035,51.313,61.945,-176.2551,25.2832,0.0000
C00847=-39.736,54.260,63.612,179.8766,0.2159,0.0000
C00848=-42.239,58.063,65.929,-177.6829,-3.4831,0.0000
C00849=-45.816,62.906,68.324,-176.4873,-5.0494,0.0000
C00850=-49.842,68.316,70.157,-175.7735,-6.1039,0.0000
C00851=-53.356,73.536,71.060,-176.9938,-6.7981,0.0000
C00852=-54.130,79.138,71.535,179.3164,-4.6272,0.0000
C00853=-51.936,84.362,71.920,178.6067,-1.8290,0.0000
C00854=-47.191,88.127,72.309,179.8678,-0.0719,0.0000
C00855=-41.335,91.053,72.565,179.9837,-0.0074,0.0000
C00856=-35.156,93.612,72.565,179.9833,-0.0062,0.0000
C00857=-28.946,95.684,72.309,179.8557,-0.0426,0.0000
C00858=-22.929,96.378,71.920,177.7221,0.3083,0.0000
C00859=-17.683,94.235,71.535,176.2430,2.7934,0.0000
C00860=-14.270,89.726,71.060,177.3000,6.9235,0.0000
C00861=-13.063,83.550,70.157,178.6617,7.2870,0.0000
C00862=-12.084,76.878,68.324,178.9074,6.0442,0.0000
C00863=-11.189,70.924,65.929,179.1735,4.0983,0.0000
C00864=-10.270,66.465,63.612,-179.9346,-0.2399,0.0000
C00865=-8.682,63.886,61.945,-159.1793,-16.0512,0.0000
C00866=-5.367,63.268,61.285,-143.6894,-2.4402,0.0000
C00867=-2.450,63.381,61.257,-143.0198,1.9701,0.0000
C00868=0.000,63.425,61.276,-143.0012,-0.0007,0.0000
C00869=0.000,62.111,63.041,-143.6741,-0.0008,0.0000
C00870=2.330,62.072,63.021,-143.6912,-1.8775,0.0000
C00871=5.165,61.970,63.050,-144.4274,2.7476,0.0000
C00872=8.436,62.639,63.741,-160.6258,15.7082,0.0000
C00873=9.975,65.350,65.485,179.9114,-0.3487,0.0000
C00874=10.861,70.011,67.904,179.1939,-4.2042,0.0000
C00875=11.743,76.212,70.393,178.9773,-5.9076,0.0000
C00876=12.712,83.133,72.289,178.7756,-7.0021,0.0000
C00877=13.898,89.524,73.219,177.5056,-6.6475,0.0000
C00878=17.338,94.193,73.707,176.4305,-2.7219,0.0000
C00879=22.659,96.427,74.103,177.8254,-0.3086,0.0000
C00880=28.778,95.739,74.502,179.8617,0.0408,0.0000
C00881=35.099,93.634,74.765,179.9840,0.0060,0.0000
C00882=41.391,91.028,74.765,179.9845,0.0071,0.0000
C00883=47.349,88.047,74.502,179.8733,0.0690,0.0000
C00884=52.162,84.206,74.103,178.6800,1.7561,0.0000
C00885=54.344,78.865,73.707,179.3988,4.4445,0.0000
C00886=53.475,73.130,73.219,-177.0458,6.4591,0.0000
C00887=49.795,67.773,72.289,-175.8969,5.8218,0.0000
C00888=45.586,62.194,70.393,-176.5353,4.9034,0.0000
C00889=41.825,57.185,67.904,-177.5933,3.5437,0.0000
C00890=39.156,53.262,65.485,-179.8161,0.3093,0.0000
C00891=38.328,50.258,63.741,-177.1498,-24.1096,0.0000
C00892=40.167,47.472,63.050,-154.7424,-28.3541,0.0000
C00893=42.244,45.539,63.021,-151.5083,-26.4003,0.0000
C00894=43.919,43.919,63.041,-152.5290,-27.4701,0.0000
C00895=45.539,42.244,63.021,-153.6002,-28.4922,0.0000
C00896=47.472,40.167,63.050,-151.6449,-25.2554,0.0000
C00897=50.258,38.328,63.741,-155.8906,-2.8500,0.0000
C00898=53.262,39.156,65.485,179.6907,-0.1839,0.0000
C00899=57.185,41.825,67.904,176.4563,-2.4067,0.0000
C00900=62.194,45.586,70.393,175.0966,-3.4647,0.0000
C00901=67.773,49.795,72.289,174.1782,-4.1031,0.0000
C00902=73.130,53.475,73.219,173.5409,-2.9542,0.0000
C00903=78.865,54.344,73.707,175.5555,0.6012,0.0000
C00904=84.206,52.162,74.103,178.2439,1.3200,0.0000
C00905=88.047,47.349,74.502,179.9310,0.1267,0.0000
C00906=91.028,41.391,74.765,179.9929,0.0155,0.0000
C00907=93.634,35.099,74.765,179.9940,0.0160,0.0000
C00908=95.739,28.778,74.502,179.9592,0.1383,0.0000
C00909=96.427,22.659,74.103,-179.6914,2.1746,0.0000
C00910=94.193,17.338,73.707,-177.2781,3.5695,0.0000
C00911=89.524,13.898,73.219,-173.3525,2.4944,0.0000
C00912=83.133,12.712,72.289,-172.9979,1.2244,0.0000
C00913=76.212,11.743,70.393,-174.0924,1.0227,0.0000
C00914=70.011,10.861,67.904,-175.7958,0.8061,0.0000
C00915=65.350,9.975,65.485,-179.6513,0.0886,0.0000
C00916=62.639,8.436,63.741,164.2918,-19.3742,0.0000
C00917=61.970,5.165,63.050,177.2524,-35.5726,0.0000
C00918=62.072,2.330,63.021,-178.1225,-36.3088,0.0000
C00919=62.111,0.000,63.041,-179.9992,-36.3259,0.0000
C00920=62.072,-2.330,63.021,178.1217,-36.3088,0.0000
C00921=61.970,-5.165,63.050,-177.2496,-35.5720,0.0000
C00922=62.640,-8.436,63.741,-164.2918,-19.3740,0.0000
C00923=65.350,-9.975,65.485,179.6513,0.0886,0.0000
C00924=70.011,-10.861,67.904,175.7958,0.8061,0.0000
C00925=76.212,-11.743,70.393,174.0924,1.0227,0.0000
C00926=83.133,-12.712,72.289,172.9979,1.2244,0.0000
C00927=89.524,-13.898,73.219,173.3525,2.4944,0.0000
C00928=94.193,-17.338,73.707,177.2781,3.5695,0.0000
C00929=96.427,-22.659,74.103,179.6914,2.1746,0.0000
C00930=95.739,-28.778,74.502,-179.9592,0.1383,0.0000
C00931=93.634,-35.099,74.765,-179.9940,0.0160,0.0000
C00932=91.028,-41.391,74.765,-179.9929,0.0155,0.0000
C00933=88.047,-47.349,74.502,-179.9310,0.1267,0.0000
C00934=84.206,-52.162,74.103,-178.2439,1.3200,0.0000
C00935=78.865,-54.344,73.707,-175.5555,0.6012,0.0000
C00936=73.130,-53.475,73.219,-173.5409,-2.9542,0.0000
C00937=67.773,-49.795,72.289,-174.1782,-4.1031,0.0000
C00938=62.194,-45.586,70.393,-175.0966,-3.4647,0.0000
C00939=57.185,-41.825,67.904,-176.4563,-2.4067,0.0000
C00940=53.262,-39.156,65.485,-179.6907,-0.1839,0.0000
C00941=50.258,-38.328,63.741,155.8904,-2.8502,0.0000
C00942=47.472,-40.167,63.050,151.6459,-25.2576,0.0000
C00943=45.539,-42.244,63.021,153.5997,-28.4917,0.0000
C00944=43.919,-43.919,63.041,152.5299,-27.4710,0.0000
C00945=42.244,-45.539,63.021,151.5078,-26.3998,0.0000
C00946=40.167,-47.472,63.050,154.7446,-28.3551,0.0000
C00947=38.328,-50.258,63.741,177.1500,-24.1094,0.0000
C00948=39.156,-53.262,65.485,179.8161,0.3093,0.0000
C00949=41.825,-57.185,67.904,177.5933,3.5437,0.0000
C00950=45.586,-62.194,70.393,176.5353,4.9034,0.0000
C00951=49.795,-67.773,72.289,175.8969,5.8218,0.0000
C00952=53.475,-73.130,73.219,177.0458,6.4591,0.0000
C00953=54.344,-78.865,73.707,-179.3988,4.4445,0.0000
C00954=52.162,-84.206,74.103,-178.6800,1.7561,0.0000
C00955=47.349,-88.047,74.502,-179.8733,0.0690,0.0000
C00956=41.391,-91.028,74.765,-179.9845,0.0071,0.0000
C00957=35.099,-93.634,74.765,-179.9840,0.0060,0.0000
C00958=28.778,-95.739,74.502,-179.8617,0.0408,0.0000
C00959=22.659,-96.427,74.103,-177.8254,-0.3086,0.0000
C00960=17.338,-94.193,73.707,-176.4305,-2.7219,0.0000
C00961=13.898,-89.524,73.219,-177.5056,-6.6475,0.0000
C00962=12.712,-83.133,72.289,-178.7756,-7.0021,0.0000
C00963=11.743,-76.212,70.393,-178.9773,-5.9076,0.0000
C00964=10.861,-70.011,67.904,-179.1939,-4.2042,0.0000
C00965=9.975,-65.350,65.485,-179.9114,-0.3487,0.0000
C00966=8.436,-62.639,63.741,160.6258,15.7082,0.0000
C00967=5.165,-61.970,63.050,144.4274,2.7476,0.0000
C00968=2.330,-62.072,63.021,143.6912,-1.8775,0.0000
C00969=0.000,-62.111,63.041,143.6741,-0.0008,0.0000
C00970=0.000,-62.111,63.041,143.6741,-0.0008,0.0000
C00971=-2.330,-62.072,63.021,143.6912,1.8783,0.0000
C00972=-5.165,-61.970,63.050,144.4280,-2.7504,0.0000
C00973=-8.436,-62.640,63.741,160.6260,-15.7082,0.0000
C00974=-9.975,-65.350,65.485,-179.9114,0.3487,0.0000
C00975=-10.861,-70.011,67.904,-179.1939,4.2042,0.0000
C00976=-11.743,-76.212,70.393,-178.9773,5.9076,0.0000
C00977=-12.712,-83.133,72.289,-178.7756,7.0021,0.0000
C00978=-13.898,-89.524,73.219,-177.5056,6.6475,0.0000
C00979=-17.338,-94.193,73.707,-176.4305,2.7219,0.0000
C00980=-22.659,-96.427,74.103,-177.8254,0.3086,0.0000
C00981=-28.778,-95.739,74.502,-179.8617,-0.0408,0.0000
C00982=-35.099,-93.634,74.765,-179.9840,-0.0060,0.0000
C00983=-41.391,-91.028,74.765,-179.9845,-0.0071,0.0000
C00984=-47.349,-88.047,74.502,-179.8733,-0.0690,0.0000
C00985=-52.162,-84.206,74.103,-178.6800,-1.7561,0.0000
C00986=-54.344,-78.865,73.707,-179.3988,-4.4445,0.0000
C00987=-53.475,-73.130,73.219,177.0458,-6.4591,0.0000
C00988=-49.795,-67.773,72.289,175.8969,-5.8218,0.0000
C00989=-45.586,-62.194,70.393,176.5353,-4.9034,0.0000
C00990=-41.825,-57.185,67.904,177.5933,-3.5437,0.0000
C00991=-39.156,-53.262,65.485,179.8161,-0.3093,0.0000
C00992=-38.328,-50.258,63.741,177.1498,24.1096,0.0000
C00993=-40.167,-47.472,63.050,154.7424,28.3541,0.0000
C00994=-42.244,-45.539,63.021,151.5083,26.4003,0.0000
C00995=-43.919,-43.919,63.041,152.5290,27.4701,0.0000
C00996=-45.539,-42.244,63.021,153.6002,28.4922,0.0000
C00997=-47.472,-40.167,63.050,151.6449,25.2554,0.0000
C00998=-50.258,-38.328,63.741,155.8906,2.8500,0.0000
C00999=-53.262,-39.156,65.485,-179.6907,0.1839,0.0000
C01000=-57.185,-41.825,67.904,-176.4563,2.4067,0.0000
C01001=-62.194,-45.586,70.393,-175.0966,3.4647,0.0000
C01002=-67.773,-49.795,72.289,-174.1782,4.1031,0.0000
C01003=-73.130,-53.475,73.219,-173.5409,2.9542,0.0000
C01004=-78.865,-54.344,73.707,-175.5555,-0.6012,0.0000
C01005=-84.206,-52.162,74.103,-178.2439,-1.3200,0.0000
C01006=-88.047,-47.349,74.502,-179.9310,-0.1267,0.0000
C01007=-91.028,-41.391,74.765,-179.9929,-0.0155,0.0000
C01008=-93.634,-35.099,74.765,-179.9940,-0.0160,0.0000
C01009=-95.739,-28.778,74.502,-179.9592,-0.1383,0.0000
C01010=-96.427,-22.659,74.103,179.6914,-2.1746,0.0000
C01011=-94.193,-17.338,73.707,177.2781,-3.5695,0.0000
C01012=-89.524,-13.898,73.219,173.3525,-2.4944,0.0000
C01013=-83.133,-12.712,72.289,172.9979,-1.2244,0.0000
C01014=-76.212,-11.743,70.393,174.0924,-1.0227,0.0000
C01015=-70.011,-10.861,67.904,175.7958,-0.8061,0.0000
C01016=-65.350,-9.975,65.485,179.6513,-0.0886,0.0000
C01017=-62.639,-8.436,63.741,-164.2918,19.3742,0.0000
C01018=-61.970,-5.165,63.050,-177.2524,35.5726,0.0000
C01019=-62.072,-2.330,63.021,178.1225,36.3088,0.0000
C01020=-62.111,0.000,63.041,179.9992,36.3259,0.0000
C01021=-62.072,2.330,63.021,-178.1217,36.3088,0.0000
C01022=-61.970,5.165,63.050,177.2496,35.5720,0.0000
C01023=-62.640,8.436,63.741,164.2918,19.3740,0.0000
C01024=-65.350,9.975,65.485,-179.6513,-0.0886,0.0000
C01025=-70.011,10.861,67.904,-175.7958,-0.8061,0.0000
C01026=-76.212,11.743,70.393,-174.0924,-1.0227,0.0000
C01027=-83.133,12.712,72.289,-172.9979,-1.2244,0.0000
C01028=-89.524,13.898,73.219,-173.3525,-2.4944,0.0000
C01029=-94.193,17.338,73.707,-177.2781,-3.5695,0.0000
C01030=-96.427,22.659,74.103,-179.6914,-2.1746,0.0000
C01031=-95.739,28.778,74.502,179.9592,-0.1383,0.0000
C01032=-93.634,35.099,74.765,179.9940,-0.0160,0.0000
C01033=-91.028,41.391,74.765,179.9929,-0.0155,0.0000
C01034=-88.047,47.349,74.502,179.9310,-0.1267,0.0000
C01035=-84.206,52.162,74.103,178.2439,-1.3200,0.0000
C01036=-78.865,54.344,73.707,175.5555,-0.6012,0.0000
C01037=-73.130,53.475,73.219,173.5409,2.9542,0.0000
C01038=-67.773,49.795,72.289,174.1782,4.1031,0.0000
C01039=-62.194,45.586,70.393,175.0966,3.4647,0.0000
C01040=-57.185,41.825,67.904,176.4563,2.4067,0.0000
C01041=-53.262,39.156,65.485,179.6907,0.1839,0.0000
C01042=-50.258,38.328,63.741,-155.8904,2.8502,0.0000
C01043=-47.472,40.167,63.050,-151.6459,25.2576,0.0000
C01044=-45.539,42.244,63.021,-153.5997,28.4917,0.0000
C01045=-43.919,43.919,63.041,-152.5299,27.4710,0.0000
C01046=-42.244,45.539,63.021,-151.5078,26.3998,0.0000
C01047=-40.167,47.472,63.050,-154.7446,28.3551,0.0000
C01048=-38.328,50.258,63.741,-177.1500,24.1094,0.0000
C01049=-39.156,53.262,65.485,-179.8161,-0.3093,0.0000
C01050=-41.825,57.185,67.904,-177.5933,-3.5437,0.0000
C01051=-45.586,62.194,70.393,-176.5353,-4.9034,0.0000
C01052=-49.795,67.773,72.289,-175.8969,-5.8218,0.0000
C01053=-53.475,73.130,73.219,-177.0458,-6.4591,0.0000
C01054=-54.344,78.865,73.707,179.3988,-4.4445,0.0000
C01055=-52.162,84.206,74.103,178.6800,-1.7561,0.0000
C01056=-47.349,88.047,74.502,179.8733,-0.0690,0.0000
C01057=-41.391,91.028,74.765,179.9845,-0.0071,0.0000
C01058=-35.099,93.634,74.765,179.9840,-0.0060,0.0000
C01059=-28.778,95.739,74.502,179.8617,-0.0408,0.0000
C01060=-22.659,96.427,74.103,177.8254,0.3086,0.0000
C01061=-17.338,94.193,73.707,176.4305,2.7219,0.0000
C01062=-13.898,89.524,73.219,177.5056,6.6475,0.0000
C01063=-12.712,83.133,72.289,178.7756,7.0021,0.0000
C01064=-11.743,76.212,70.393,178.9773,5.9076,0.0000
C01065=-10.861,70.011,67.904,179.1939,4.2042,0.0000
C01066=-9.975,65.350,65.485,179.9114,0.3487,0.0000
C01067=-8.436,62.640,63.741,-160.6260,-15.7082,0.0000
C01068=-5.165,61.970,63.050,-144.4280,-2.7504,0.0000
C01069=-2.330,62.072,63.021,-143.6912,1.8783,0.0000
C01070=0.000,62.111,63.041,-143.6741,-0.0008,0.0000
C01071=0.000,60.820,64.822,-144.4513,-0.0008,0.0000
C01072=2.212,60.785,64.801,-144.4668,-1.7783,0.0000
C01073=4.967,60.695,64.832,-145.2737,3.0327,0.0000
C01074=8.195,61.417,65.554,-162.0706,15.2576,0.0000
C01075=9.686,64.262,67.375,179.7975,-0.8529,0.0000
C01076=10.544,69.129,69.894,179.2239,-4.2461,0.0000
C01077=11.418,75.576,72.474,179.0505,-5.7116,0.0000
C01078=12.382,82.740,74.428,178.8887,-6.6531,0.0000
C01079=13.550,89.334,75.383,177.7173,-6.3021,0.0000
C01080=17.016,94.154,75.883,176.6505,-2.6124,0.0000
C01081=22.407,96.473,76.288,177.9510,-0.3030,0.0000
C01082=28.621,95.791,76.696,179.8693,0.0384,0.0000
C01083=35.046,93.654,76.964,179.9850,0.0056,0.0000
C01084=41.442,91.005,76.964,179.9854,0.0067,0.0000
C01085=47.497,87.973,76.696,179.8804,0.0653,0.0000
C01086=52.372,84.060,76.288,178.7650,1.6633,0.0000
C01087=54.545,78.609,75.883,179.4774,4.2121,0.0000
C01088=53.588,72.750,75.383,-177.1430,6.0665,0.0000
C01089=49.751,67.261,74.428,-176.0664,5.4947,0.0000
C01090=45.367,61.514,72.474,-176.6232,4.7129,0.0000
C01091=41.426,56.337,69.894,-177.5424,3.5522,0.0000
C01092=38.591,52.289,67.375,-179.5401,0.7463,0.0000
C01093=37.634,49.223,65.554,-177.9435,-22.8637,0.0000
C01094=39.406,46.429,64.832,-155.6464,-27.8147,0.0000
C01095=41.417,44.545,64.801,-152.2131,-25.7824,0.0000
C01096=43.006,43.006,64.822,-153.1928,-26.8062,0.0000
C01097=44.545,41.417,64.801,-154.2181,-27.7874,0.0000
C01098=46.430,39.405,64.832,-152.1844,-24.3513,0.0000
C01099=49.223,37.634,65.554,-157.1366,-2.0563,0.0000
C01100=52.289,38.591,67.375,179.2537,-0.4599,0.0000
C01101=56.337,41.426,69.894,176.4478,-2.4576,0.0000
C01102=61.514,45.367,72.474,175.2871,-3.3768,0.0000
C01103=67.261,49.751,74.428,174.5053,-3.9336,0.0000
C01104=72.750,53.588,75.383,173.9335,-2.8570,0.0000
C01105=78.609,54.545,75.883,175.7879,0.5226,0.0000
C01106=84.060,52.372,76.288,178.3367,1.2350,0.0000
C01107=87.973,47.497,76.696,179.9347,0.1196,0.0000
C01108=91.005,41.442,76.964,179.9933,0.0146,0.0000
C01109=93.654,35.046,76.964,179.9944,0.0150,0.0000
C01110=95.791,28.621,76.696,179.9616,0.1307,0.0000
C01111=96.473,22.407,76.288,-179.6970,2.0490,0.0000
C01112=94.154,17.016,75.883,-177.3876,3.3495,0.0000
C01113=89.334,13.550,75.383,-173.6979,2.2827,0.0000
C01114=82.740,12.382,74.428,-173.3469,1.1113,0.0000
C01115=75.576,11.418,72.474,-174.2884,0.9495,0.0000
C01116=69.129,10.544,69.894,-175.7539,0.7761,0.0000
C01117=64.262,9.686,67.375,-179.1471,0.2025,0.0000
C01118=61.417,8.195,65.554,164.7424,-17.9294,0.0000
C01119=60.695,4.967,64.832,176.9673,-34.7263,0.0000
C01120=60.785,2.212,64.801,-178.2217,-35.5332,0.0000
C01121=60.820,0.000,64.822,-179.9992,-35.5487,0.0000
C01122=60.785,-2.212,64.801,178.2207,-35.5333,0.0000
C01123=60.695,-4.967,64.832,-176.9646,-34.7257,0.0000
C01124=61.417,-8.195,65.554,-164.7424,-17.9290,0.0000
C01125=64.262,-9.686,67.375,179.1471,0.2025,0.0000
C01126=69.129,-10.544,69.894,175.7539,0.7761,0.0000
C01127=75.576,-11.418,72.474,174.2884,0.9495,0.0000
C01128=82.740,-12.382,74.428,173.3469,1.1113,0.0000
C01129=89.334,-13.550,75.383,173.6979,2.2827,0.0000
C01130=94.154,-17.016,75.883,177.3876,3.3495,0.0000
C01131=96.473,-22.407,76.288,179.6970,2.0490,0.0000
C01132=95.791,-28.621,76.696,-179.9616,0.1307,0.0000
C01133=93.654,-35.046,76.964,-179.9944,0.0150,0.0000
C01134=91.005,-41.442,76.964,-179.9933,0.0146,0.0000
C01135=87.973,-47.497,76.696,-179.9347,0.1196,0.0000
C01136=84.060,-52.372,76.288,-178.3367,1.2350,0.0000
C01137=78.609,-54.545,75.883,-175.7879,0.5226,0.0000
C01138=72.750,-53.588,75.383,-173.9335,-2.8570,0.0000
C01139=67.261,-49.751,74.428,-174.5053,-3.9336,0.0000
C01140=61.514,-45.367,72.474,-175.2871,-3.3768,0.0000
C01141=56.337,-41.426,69.894,-176.4478,-2.4576,0.0000
C01142=52.289,-38.591,67.375,-179.2537,-0.4599,0.0000
C01143=49.223,-37.634,65.554,157.1363,-2.0565,0.0000
C01144=46.429,-39.406,64.832,152.1853,-24.3536,0.0000
C01145=44.545,-41.417,64.801,154.2176,-27.7869,0.0000
C01146=43.006,-43.006,64.822,153.1938,-26.8072,0.0000
C01147=41.417,-44.545,64.801,152.2126,-25.7819,0.0000
C01148=39.405,-46.430,64.832,155.6487,-27.8156,0.0000
C01149=37.634,-49.223,65.554,177.9437,-22.8634,0.0000
C01150=38.591,-52.289,67.375,179.5401,0.7463,0.0000
C01151=41.426,-56.337,69.894,177.5424,3.5522,0.0000
C01152=45.367,-61.514,72.474,176.6232,4.7129,0.0000
C01153=49.751,-67.261,74.428,176.0664,5.4947,0.0000
C01154=53.588,-72.750,75.383,177.1430,6.0665,0.0000
C01155=54.545,-78.609,75.883,-179.4774,4.2121,0.0000
C01156=52.372,-84.060,76.288,-178.7650,1.6633,0.0000
C01157=47.497,-87.973,76.696,-179.8804,0.0653,0.0000
C01158=41.442,-91.005,76.964,-179.9854,0.0067,0.0000
C01159=35.046,-93.654,76.964,-179.9850,0.0056,0.0000
C01160=28.621,-95.791,76.696,-179.8693,0.0384,0.0000
C01161=22.407,-96.473,76.288,-177.9510,-0.3030,0.0000
C01162=17.016,-94.154,75.883,-176.6505,-2.6124,0.0000
C01163=13.550,-89.334,75.383,-177.7173,-6.3021,0.0000
C01164=12.382,-82.740,74.428,-178.8887,-6.6531,0.0000
C01165=11.418,-75.576,72.474,-179.0505,-5.7116,0.0000
C01166=10.544,-69.129,69.894,-179.2239,-4.2461,0.0000
C01167=9.686,-64.262,67.375,-179.7975,-0.8529,0.0000
C01168=8.195,-61.417,65.554,162.0706,15.2576,0.0000
C01169=4.967,-60.695,64.832,145.2737,3.0327,0.0000
C01170=2.212,-60.785,64.801,144.4668,-1.7783,0.0000
C01171=0.000,-60.820,64.822,144.4513,-0.0008,0.0000
C01172=0.000,-60.820,64.822,144.4513,-0.0008,0.0000
C01173=-2.212,-60.785,64.801,144.4667,1.7793,0.0000
C01174=-4.967,-60.695,64.832,145.2743,-3.0354,0.0000
C01175=-8.195,-61.417,65.554,162.0710,-15.2576,0.0000
C01176=-9.686,-64.262,67.375,-179.7975,0.8529,0.0000
C01177=-10.544,-69.129,69.894,-179.2239,4.2461,0.0000
C01178=-11.418,-75.576,72.474,-179.0505,5.7116,0.0000
C01179=-12.382,-82.740,74.428,-178.8887,6.6531,0.0000
C01180=-13.550,-89.334,75.383,-177.7173,6.3021,0.0000
C01181=-17.016,-94.154,75.883,-176.6505,2.6124,0.0000
C01182=-22.407,-96.473,76.288,-177.9510,0.3030,0.0000
C01183=-28.621,-95.791,76.696,-179.8693,-0.0384,0.0000
C01184=-35.046,-93.654,76.964,-179.9850,-0.0056,0.0000
C01185=-41.442,-91.005,76.964,-179.9854,-0.0067,0.0000
C01186=-47.497,-87.973,76.696,-179.8804,-0.0653,0.0000
C01187=-52.372,-84.060,76.288,-178.7650,-1.6633,0.0000
C01188=-54.545,-78.609,75.883,-179.4774,-4.2121,0.0000
C01189=-53.588,-72.750,75.383,177.1430,-6.0665,0.0000
C01190=-49.751,-67.261,74.428,176.0664,-5.4947,0.0000
C01191=-45.367,-61.514,72.474,176.6232,-4.7129,0.0000
C01192=-41.426,-56.337,69.894,177.5424,-3.5522,0.0000
C01193=-38.591,-52.289,67.375,179.5401,-0.7463,0.0000
C01194=-37.634,-49.223,65.554,177.9435,22.8637,0.0000
C01195=-39.406,-46.429,64.832,155.6464,27.8147,0.0000
C01196=-41.417,-44.545,64.801,152.2131,25.7824,0.0000
C01197=-43.006,-43.006,64.822,153.1928,26.8062,0.0000
C01198=-44.545,-41.417,64.801,154.2181,27.7874,0.0000
C01199=-46.430,-39.405,64.832,152.1844,24.3513,0.0000
C01200=-49.223,-37.634,65.554,157.1366,2.0563,0.0000
C01201=-52.289,-38.591,67.375,-179.2537,0.4599,0.0000
C01202=-56.337,-41.426,69.894,-176.4478,2.4576,0.0000
C01203=-61.514,-45.367,72.474,-175.2871,3.3768,0.0000
C01204=-67.261,-49.751,74.428,-174.5053,3.9336,0.0000
C01205=-72.750,-53.588,75.383,-173.9335,2.8570,0.0000
C01206=-78.609,-54.545,75.883,-175.7879,-0.5226,0.0000
C01207=-84.060,-52.372,76.288,-178.3367,-1.2350,0.0000
C01208=-87.973,-47.497,76.696,-179.9347,-0.1196,0.0000
C01209=-91.005,-41.442,76.964,-179.9933,-0.0146,0.0000
C01210=-93.654,-35.046,76.964,-179.9944,-0.0150,0.0000
C01211=-95.791,-28.621,76.696,-179.9616,-0.1307,0.0000
C01212=-96.473,-22.407,76.288,179.6970,-2.0490,0.0000
C01213=-94.154,-17.016,75.883,177.3876,-3.3495,0.0000
C01214=-89.334,-13.550,75.383,173.6979,-2.2827,0.0000
C01215=-82.740,-12.382,74.428,173.3469,-1.1113,0.0000
C01216=-75.576,-11.418,72.474,174.2884,-0.9495,0.0000
C01217=-69.129,-10.544,69.894,175.7539,-0.7761,0.0000
C01218=-64.262,-9.686,67.375,179.1471,-0.2025,0.0000
C01219=-61.417,-8.195,65.554,-164.7424,17.9294,0.0000
C01220=-60.695,-4.967,64.832,-176.9673,34.7263,0.0000
C01221=-60.785,-2.212,64.801,178.2217,35.5332,0.0000
C01222=-60.820,0.000,64.822,179.9992,35.5487,0.0000
C01223=-60.785,2.212,64.801,-178.2207,35.5333,0.0000
C01224=-60.695,4.967,64.832,176.9646,34.7257,0.0000
C01225=-61.417,8.195,65.554,164.7424,17.9290,0.0000
C01226=-64.262,9.686,67.375,-179.1471,-0.2025,0.0000
C01227=-69.129,10.544,69.894,-175.7539,-0.7761,0.0000
C01228=-75.576,11.418,72.474,-174.2884,-0.9495,0.0000
C01229=-82.740,12.382,74.428,-173.3469,-1.1113,0.0000
C01230=-89.334,13.550,75.383,-173.6979,-2.2827,0.0000
C01231=-94.154,17.016,75.883,-177.3876,-3.3495,0.0000
C01232=-96.473,22.407,76.288,-179.6970,-2.0490,0.0000
C01233=-95.791,28.621,76.696,179.9616,-0.1307,0.0000
C01234=-93.654,35.046,76.964,179.9944,-0.0150,0.0000
C01235=-91.005,41.442,76.964,179.9933,-0.0146,0.0000
C01236=-87.973,47.497,76.696,179.9347,-0.1196,0.0000
C01237=-84.060,52.372,76.288,178.3367,-1.2350,0.0000
C01238=-78.609,54.545,75.883,175.7879,-0.5226,0.0000
C01239=-72.750,53.588,75.383,173.9335,2.8570,0.0000
C01240=-67.261,49.751,74.428,174.5053,3.9336,0.0000
C01241=-61.514,45.367,72.474,175.2871,3.3768,0.0000
C01242=-56.337,41.426,69.894,176.4478,2.4576,0.0000
C01243=-52.289,38.591,67.375,179.2537,0.4599,0.0000
C01244=-49.223,37.634,65.554,-157.1363,2.0565,0.0000
C01245=-46.429,39.406,64.832,-152.1853,24.3536,0.0000
C01246=-44.545,41.417,64.801,-154.2176,27.7869,0.0000
C01247=-43.006,43.006,64.822,-153.1938,26.8072,0.0000
C01248=-41.417,44.545,64.801,-152.2126,25.7819,0.0000
C01249=-39.405,46.430,64.832,-155.6487,27.8156,0.0000
C01250=-37.634,49.223,65.554,-177.9437,22.8634,0.0000
C01251=-38.591,52.289,67.375,-179.5401,-0.7463,0.0000
C01252=-41.426,56.337,69.894,-177.5424,-3.5522,0.0000
C01253=-45.367,61.514,72.474,-176.6232,-4.7129,0.0000
C01254=-49.751,67.261,74.428,-176.0664,-5.4947,0.0000
C01255=-53.588,72.750,75.383,-177.1430,-6.0665,0.0000
C01256=-54.545,78.609,75.883,179.4774,-4.2121,0.0000
C01257=-52.372,84.060,76.288,178.7650,-1.6633,0.0000
C01258=-47.497,87.973,76.696,179.8804,-0.0653,0.0000
C01259=-41.442,91.005,76.964,179.9854,-0.0067,0.0000
C01260=-35.046,93.654,76.964,179.9850,-0.0056,0.0000
C01261=-28.621,95.791,76.696,179.8693,-0.0384,0.0000
C01262=-22.407,96.473,76.288,177.9510,0.3030,0.0000
C01263=-17.016,94.154,75.883,176.6505,2.6124,0.0000
C01264=-13.550,89.334,75.383,177.7173,6.3021,0.0000
C01265=-12.382,82.740,74.428,178.8887,6.6531,0.0000
C01266=-11.418,75.576,72.474,179.0505,5.7116,0.0000
C01267=-10.544,69.129,69.894,179.2239,4.2461,0.0000
C01268=-9.686,64.262,67.375,179.7975,0.8529,0.0000
C01269=-8.195,61.417,65.554,-162.0710,-15.2576,0.0000
C01270=-4.967,60.695,64.832,-145.2743,-3.0354,0.0000
C01271=-2.212,60.785,64.801,-144.4667,1.7793,0.0000
C01272=0.000,60.820,64.822,-144.4513,-0.0008,0.0000
C01273=0.000,59.554,66.621,-145.3415,-0.0009,0.0000
C01274=2.097,59.523,66.599,-145.3553,-1.6722,0.0000
C01275=4.772,59.445,66.632,-146.2352,3.2869,0.0000
C01276=7.959,60.221,67.386,-163.5021,14.7072,0.0000
C01277=9.406,63.206,69.285,179.7171,-1.2730,0.0000
C01278=10.239,68.282,71.901,179.2620,-4.2251,0.0000
C01279=11.109,74.974,74.567,179.1263,-5.4571,0.0000
C01280=12.073,82.372,76.575,179.0007,-6.2410,0.0000
C01281=13.226,89.158,77.551,177.9343,-5.8891,0.0000
C01282=16.717,94.118,78.062,176.9018,-2.4653,0.0000
C01283=22.174,96.515,78.476,178.0988,-0.2913,0.0000
C01284=28.477,95.839,78.891,179.8785,0.0356,0.0000
C01285=34.998,93.673,79.163,179.9861,0.0052,0.0000
C01286=41.489,90.984,79.163,179.9865,0.0062,0.0000
C01287=47.632,87.904,78.891,179.8889,0.0607,0.0000
C01288=52.567,83.926,78.476,178.8613,1.5505,0.0000
C01289=54.731,78.373,78.062,179.5514,3.9310,0.0000
C01290=53.692,72.396,77.551,-177.2844,5.6222,0.0000
C01291=49.709,66.782,76.575,-176.2813,5.1235,0.0000
C01292=45.159,60.870,74.567,-176.7508,4.4791,0.0000
C01293=41.042,55.523,71.901,-177.5304,3.5105,0.0000
C01294=38.042,51.344,69.285,-179.2998,1.1002,0.0000
C01295=36.955,48.211,67.386,-178.6352,-21.5554,0.0000
C01296=38.660,45.408,66.632,-156.6295,-27.1736,0.0000
C01297=40.607,43.572,66.599,-153.0121,-25.0783,0.0000
C01298=42.111,42.111,66.621,-153.9470,-26.0519,0.0000
C01299=43.571,40.607,66.599,-154.9223,-26.9884,0.0000
C01300=45.409,38.659,66.632,-152.8255,-23.3682,0.0000
C01301=48.211,36.955,67.386,-158.4450,-1.3645,0.0000
C01302=51.344,38.042,69.285,178.8998,-0.7002,0.0000
C01303=55.523,41.042,71.901,176.4895,-2.4696,0.0000
C01304=60.870,45.159,74.567,175.5209,-3.2492,0.0000
C01305=66.782,49.709,76.575,174.8765,-3.7187,0.0000
C01306=72.396,53.692,77.551,174.3778,-2.7156,0.0000
C01307=78.373,54.731,78.062,176.0690,0.4486,0.0000
C01308=83.926,52.567,78.476,178.4495,1.1387,0.0000
C01309=87.904,47.632,78.891,179.9393,0.1111,0.0000
C01310=90.984,41.489,79.163,179.9938,0.0135,0.0000
C01311=93.673,34.998,79.163,179.9948,0.0139,0.0000
C01312=95.839,28.477,78.891,179.9644,0.1215,0.0000
C01313=96.515,22.174,78.476,-179.7087,1.9012,0.0000
C01314=94.118,16.717,78.062,-177.5347,3.0982,0.0000
C01315=89.158,13.226,77.551,-174.1109,2.0657,0.0000
C01316=82.372,12.073,76.575,-173.7590,0.9993,0.0000
C01317=74.974,11.109,74.567,-174.5429,0.8737,0.0000
C01318=68.282,10.239,71.901,-175.7749,0.7380,0.0000
C01319=63.206,9.406,69.285,-178.7270,0.2829,0.0000
C01320=60.221,7.959,67.386,165.2928,-16.4979,0.0000
C01321=59.445,4.772,66.632,176.7131,-33.7648,0.0000
C01322=59.523,2.097,66.599,-178.3278,-34.6447,0.0000
C01323=59.554,0.000,66.621,-179.9991,-34.6585,0.0000
C01324=59.523,-2.096,66.599,178.3268,-34.6448,0.0000
C01325=59.445,-4.772,66.632,-176.7103,-33.7640,0.0000
C01326=60.222,-7.959,67.386,-165.2928,-16.4975,0.0000
C01327=63.206,-9.406,69.285,178.7270,0.2829,0.0000
C01328=68.282,-10.239,71.901,175.7749,0.7380,0.0000
C01329=74.974,-11.109,74.567,174.5429,0.8737,0.0000
C01330=82.372,-12.073,76.575,173.7590,0.9993,0.0000
C01331=89.158,-13.226,77.551,174.1109,2.0657,0.0000
C01332=94.118,-16.717,78.062,177.5347,3.0982,0.0000
C01333=96.515,-22.174,78.476,179.7087,1.9012,0.0000
C01334=95.839,-28.477,78.891,-179.9644,0.1215,0.0000
C01335=93.673,-34.998,79.163,-179.9948,0.0139,0.0000
C01336=90.984,-41.489,79.163,-179.9938,0.0135,0.0000
C01337=87.904,-47.632,78.891,-179.9393,0.1111,0.0000
C01338=83.926,-52.567,78.476,-178.4495,1.1387,0.0000
C01339=78.373,-54.731,78.062,-176.0690,0.4486,0.0000
C01340=72.396,-53.692,77.551,-174.3778,-2.7156,0.0000
C01341=66.782,-49.709,76.575,-174.8765,-3.7187,0.0000
C01342=60.870,-45.159,74.567,-175.5209,-3.2492,0.0000
C01343=55.523,-41.042,71.901,-176.4895,-2.4696,0.0000
C01344=51.344,-38.042,69.285,-178.8998,-0.7002,0.0000
C01345=48.211,-36.955,67.386,158.4446,-1.3648,0.0000
C01346=45.408,-38.660,66.632,152.8264,-23.3705,0.0000
C01347=43.572,-40.607,66.599,154.9217,-26.9879,0.0000
C01348=42.111,-42.111,66.621,153.9481,-26.0530,0.0000
C01349=40.607,-43.571,66.599,153.0116,-25.0777,0.0000
C01350=38.659,-45.409,66.632,156.6318,-27.1745,0.0000
C01351=36.955,-48.211,67.386,178.6355,-21.5550,0.0000
C01352=38.042,-51.344,69.285,179.2998,1.1002,0.0000
C01353=41.042,-55.523,71.901,177.5304,3.5105,0.0000
C01354=45.159,-60.870,74.567,176.7508,4.4791,0.0000
C01355=49.709,-66.782,76.575,176.2813,5.1235,0.0000
C01356=53.692,-72.396,77.551,177.2844,5.6222,0.0000
C01357=54.731,-78.373,78.062,-179.5514,3.9310,0.0000
C01358=52.567,-83.926,78.476,-178.8613,1.5505,0.0000
C01359=47.632,-87.904,78.891,-179.8889,0.0607,0.0000
C01360=41.489,-90.984,79.163,-179.9865,0.0062,0.0000
C01361=34.998,-93.673,79.163,-179.9861,0.0052,0.0000
C01362=28.477,-95.839,78.891,-179.8785,0.0356,0.0000
C01363=22.174,-96.515,78.476,-178.0988,-0.2913,0.0000
C01364=16.717,-94.118,78.062,-176.9018,-2.4653,0.0000
C01365=13.226,-89.158,77.551,-177.9343,-5.8891,0.0000
C01366=12.073,-82.372,76.575,-179.0007,-6.2410,0.0000
C01367=11.109,-74.974,74.567,-179.1263,-5.4571,0.0000
C01368=10.239,-68.282,71.901,-179.2620,-4.2251,0.0000
C01369=9.406,-63.206,69.285,-179.7171,-1.2730,0.0000
C01370=7.959,-60.221,67.386,163.5021,14.7072,0.0000
C01371=4.772,-59.445,66.632,146.2352,3.2869,0.0000
C01372=2.097,-59.523,66.599,145.3553,-1.6722,0.0000
C01373=0.000,-59.554,66.621,145.3415,-0.0009,0.0000
C01374=0.000,-59.554,66.621,145.3415,-0.0009,0.0000
C01375=-2.096,-59.523,66.599,145.3552,1.6732,0.0000
C01376=-4.772,-59.445,66.632,146.2360,-3.2897,0.0000
C01377=-7.959,-60.222,67.386,163.5025,-14.7072,0.0000
C01378=-9.406,-63.206,69.285,-179.7171,1.2730,0.0000
C01379=-10.239,-68.282,71.901,-179.2620,4.2251,0.0000
C01380=-11.109,-74.974,74.567,-179.1263,5.4571,0.0000
C01381=-12.073,-82.372,76.575,-179.0007,6.2410,0.0000
C01382=-13.226,-89.158,77.551,-177.9343,5.8891,0.0000
C01383=-16.717,-94.118,78.062,-176.9018,2.4653,0.0000
C01384=-22.174,-96.515,78.476,-178.0988,0.2913,0.0000
C01385=-28.477,-95.839,78.891,-179.8785,-0.0356,0.0000
C01386=-34.998,-93.673,79.163,-179.9861,-0.0052,0.0000
C01387=-41.489,-90.984,79.163,-179.9865,-0.0062,0.0000
C01388=-47.632,-87.904,78.891,-179.8889,-0.0607,0.0000
C01389=-52.567,-83.926,78.476,-178.8613,-1.5505,0.0000
C01390=-54.731,-78.373,78.062,-179.5514,-3.9310,0.0000
C01391=-53.692,-72.396,77.551,177.2844,-5.6222,0.0000
C01392=-49.709,-66.782,76.575,176.2813,-5.1235,0.0000
C01393=-45.159,-60.870,74.567,176.7508,-4.4791,0.0000
C01394=-41.042,-55.523,71.901,177.5304,-3.5105,0.0000
C01395=-38.042,-51.344,69.285,179.2998,-1.1002,0.0000
C01396=-36.955,-48.211,67.386,178.6352,21.5554,0.0000
C01397=-38.660,-45.408,66.632,156.6295,27.1736,0.0000
C01398=-40.607,-43.572,66.599,153.0121,25.0783,0.0000
C01399=-42.111,-42.111,66.621,153.9470,26.0519,0.0000
C01400=-43.571,-40.607,66.599,154.9223,26.9884,0.0000
C01401=-45.409,-38.659,66.632,152.8255,23.3682,0.0000
C01402=-48.211,-36.955,67.386,158.4450,1.3645,0.0000
C01403=-51.344,-38.042,69.285,-178.8998,0.7002,0.0000
C01404=-55.523,-41.042,71.901,-176.4895,2.4696,0.0000
C01405=-60.870,-45.159,74.567,-175.5209,3.2492,0.0000
C01406=-66.782,-49.709,76.575,-174.8765,3.7187,0.0000
C01407=-72.396,-53.692,77.551,-174.3778,2.7156,0.0000
C01408=-78.373,-54.731,78.062,-176.0690,-0.4486,0.0000
C01409=-83.926,-52.567,78.476,-178.4495,-1.1387,0.0000
C01410=-87.904,-47.632,78.891,-179.9393,-0.1111,0.0000
C01411=-90.984,-41.489,79.163,-179.9938,-0.0135,0.0000
C01412=-93.673,-34.998,79.163,-179.9948,-0.0139,0.0000
C01413=-95.839,-28.477,78.891,-179.9644,-0.1215,0.0000
C01414=-96.515,-22.174,78.476,179.7087,-1.9012,0.0000
C01415=-94.118,-16.717,78.062,177.5347,-3.0982,0.0000
C01416=-89.158,-13.226,77.551,174.1109,-2.0657,0.0000
C01417=-82.372,-12.073,76.575,173.7590,-0.9993,0.0000
C01418=-74.974,-11.109,74.567,174.5429,-0.8737,0.0000
C01419=-68.282,-10.239,71.901,175.7749,-0.7380,0.0000
C01420=-63.206,-9.406,69.285,178.7270,-0.2829,0.0000
C01421=-60.221,-7.959,67.386,-165.2928,16.4979,0.0000
C01422=-59.445,-4.772,66.632,-176.7131,33.7648,0.0000
C01423=-59.523,-2.097,66.599,178.3278,34.6447,0.0000
C01424=-59.554,0.000,66.621,179.9991,34.6585,0.0000
C01425=-59.523,2.096,66.599,-178.3268,34.6448,0.0000
C01426=-59.445,4.772,66.632,176.7103,33.7640,0.0000
C01427=-60.222,7.959,67.386,165.2928,16.4975,0.0000
C01428=-63.206,9.406,69.285,-178.7270,-0.2829,0.0000
C01429=-68.282,10.239,71.901,-175.7749,-0.7380,0.0000
C01430=-74.974,11.109,74.567,-174.5429,-0.8737,0.0000
C01431=-82.372,12.073,76.575,-173.7590,-0.9993,0.0000
C01432=-89.158,13.226,77.551,-174.1109,-2.0657,0.0000
C01433=-94.118,16.717,78.062,-177.5347,-3.0982,0.0000
C01434=-96.515,22.174,78.476,-179.7087,-1.9012,0.0000
C01435=-95.839,28.477,78.891,179.9644,-0.1215,0.0000
C01436=-93.673,34.998,79.163,179.9948,-0.0139,0.0000
C01437=-90.984,41.489,79.163,179.9938,-0.0135,0.0000
C01438=-87.904,47.632,78.891,179.9393,-0.1111,0.0000
C01439=-83.926,52.567,78.476,178.4495,-1.1387,0.0000
C01440=-78.373,54.731,78.062,176.0690,-0.4486,0.0000
C01441=-72.396,53.692,77.551,174.3778,2.7156,0.0000
C01442=-66.782,49.709,76.575,174.8765,3.7187,0.0000
C01443=-60.870,45.159,74.567,175.5209,3.2492,0.0000
C01444=-55.523,41.042,71.901,176.4895,2.4696,0.0000
C01445=-51.344,38.042,69.285,178.8998,0.7002,0.0000
C01446=-48.211,36.955,67.386,-158.4446,1.3648,0.0000
C01447=-45.408,38.660,66.632,-152.8264,23.3705,0.0000
C01448=-43.572,40.607,66.599,-154.9217,26.9879,0.0000
C01449=-42.111,42.111,66.621,-153.9481,26.0530,0.0000
C01450=-40.607,43.571,66.599,-153.0116,25.0777,0.0000
C01451=-38.659,45.409,66.632,-156.6318,27.1745,0.0000
C01452=-36.955,48.211,67.386,-178.6355,21.5550,0.0000
C01453=-38.042,51.344,69.285,-179.2998,-1.1002,0.0000
C01454=-41.042,55.523,71.901,-177.5304,-3.5105,0.0000
C01455=-45.159,60.870,74.567,-176.7508,-4.4791,0.0000
C01456=-49.709,66.782,76.575,-176.2813,-5.1235,0.0000
C01457=-53.692,72.396,77.551,-177.2844,-5.6222,0.0000
C01458=-54.731,78.373,78.062,179.5514,-3.9310,0.0000
C01459=-52.567,83.926,78.476,178.8613,-1.5505,0.0000
C01460=-47.632,87.904,78.891,179.8889,-0.0607,0.0000
C01461=-41.489,90.984,79.163,179.9865,-0.0062,0.0000
C01462=-34.998,93.673,79.163,179.9861,-0.0052,0.0000
C01463=-28.477,95.839,78.891,179.8785,-0.0356,0.0000
C01464=-22.174,96.515,78.476,178.0988,0.2913,0.0000
C01465=-16.717,94.118,78.062,176.9018,2.4653,0.0000
C01466=-13.226,89.158,77.551,177.9343,5.8891,0.0000
C01467=-12.073,82.372,76.575,179.0007,6.2410,0.0000
C01468=-11.109,74.974,74.567,179.1263,5.4571,0.0000
C01469=-10.239,68.282,71.901,179.2620,4.2251,0.0000
C01470=-9.406,63.206,69.285,179.7171,1.2730,0.0000
C01471=-7.959,60.222,67.386,-163.5025,-14.7072,0.0000
C01472=-4.772,59.445,66.632,-146.2360,-3.2897,0.0000
C01473=-2.096,59.523,66.599,-145.3552,1.6732,0.0000
C01474=0.000,59.554,66.621,-145.3415,-0.0009,0.0000
C01475=0.000,58.319,68.442,-146.3550,-0.0009,0.0000
C01476=1.984,58.291,68.419,-146.3668,-1.5596,0.0000
C01477=4.582,58.225,68.453,-147.3209,3.5043,0.0000
C01478=7.730,59.058,69.238,-164.9099,14.0649,0.0000
C01479=9.135,62.185,71.215,179.6644,-1.6099,0.0000
C01480=9.949,67.473,73.927,179.3067,-4.1423,0.0000
C01481=10.820,74.409,76.674,179.2045,-5.1449,0.0000
C01482=11.787,82.032,78.729,179.1118,-5.7669,0.0000
C01483=12.929,88.996,79.725,178.1562,-5.4103,0.0000
C01484=16.445,94.085,80.245,177.1832,-2.2811,0.0000
C01485=21.964,96.553,80.665,178.2682,-0.2736,0.0000
C01486=28.347,95.882,81.086,179.8893,0.0324,0.0000
C01487=34.955,93.690,81.363,179.9874,0.0047,0.0000
C01488=41.532,90.965,81.363,179.9877,0.0056,0.0000
C01489=47.755,87.843,81.086,179.8988,0.0554,0.0000
C01490=52.743,83.804,80.665,178.9686,1.4181,0.0000
C01491=54.900,78.157,80.245,179.6205,3.6025,0.0000
C01492=53.787,72.072,79.725,-177.4688,5.1275,0.0000
C01493=49.670,66.340,78.729,-176.5407,4.7091,0.0000
C01494=44.964,60.266,76.674,-176.9177,4.2028,0.0000
C01495=40.676,54.746,73.927,-177.5576,3.4203,0.0000
C01496=37.512,50.430,71.215,-179.0987,1.3757,0.0000
C01497=36.294,47.226,69.238,-179.2260,-20.1942,0.0000
C01498=37.931,44.411,68.453,-157.6922,-26.4224,0.0000
C01499=39.816,42.621,68.419,-153.9116,-24.2820,0.0000
C01500=41.238,41.238,68.442,-154.7977,-25.2012,0.0000
C01501=42.621,39.816,68.419,-155.7185,-26.0890,0.0000
C01502=44.412,37.931,68.453,-153.5766,-22.3055,0.0000
C01503=47.226,36.294,69.238,-159.8063,-0.7736,0.0000
C01504=50.430,37.512,71.215,178.6243,-0.9013,0.0000
C01505=54.746,40.676,73.927,176.5797,-2.4424,0.0000
C01506=60.266,44.964,76.674,175.7972,-3.0823,0.0000
C01507=66.340,49.670,78.729,175.2909,-3.4593,0.0000
C01508=72.072,53.787,79.725,174.8725,-2.5312,0.0000
C01509=78.157,54.900,80.245,176.3975,0.3795,0.0000
C01510=83.804,52.743,80.665,178.5819,1.0314,0.0000
C01511=87.843,47.755,81.086,179.9446,0.1012,0.0000
C01512=90.965,41.532,81.363,179.9944,0.0123,0.0000
C01513=93.690,34.955,81.363,179.9953,0.0126,0.0000
C01514=95.882,28.347,81.086,179.9676,0.1107,0.0000
C01515=96.553,21.964,80.665,-179.7264,1.7318,0.0000
C01516=94.085,16.445,80.245,-177.7189,2.8168,0.0000
C01517=88.996,12.929,79.725,-174.5897,1.8438,0.0000
C01518=82.032,11.787,78.729,-174.2331,0.8882,0.0000
C01519=74.409,10.820,76.674,-174.8551,0.7955,0.0000
C01520=67.473,9.949,73.927,-175.8577,0.6933,0.0000
C01521=62.185,9.135,71.215,-178.3901,0.3356,0.0000
C01522=59.058,7.730,69.238,165.9351,-15.0901,0.0000
C01523=58.225,4.582,68.453,176.4957,-32.6791,0.0000
C01524=58.291,1.984,68.419,-178.4404,-33.6332,0.0000
C01525=58.319,0.000,68.442,-179.9991,-33.6450,0.0000
C01526=58.291,-1.983,68.419,178.4394,-33.6332,0.0000
C01527=58.225,-4.583,68.453,-176.4929,-32.6783,0.0000
C01528=59.058,-7.730,69.238,-165.9352,-15.0895,0.0000
C01529=62.185,-9.135,71.215,178.3901,0.3356,0.0000
C01530=67.473,-9.949,73.927,175.8577,0.6933,0.0000
C01531=74.409,-10.820,76.674,174.8551,0.7955,0.0000
C01532=82.032,-11.787,78.729,174.2331,0.8882,0.0000
C01533=88.996,-12.929,79.725,174.5897,1.8438,0.0000
C01534=94.085,-16.445,80.245,177.7189,2.8168,0.0000
C01535=96.553,-21.964,80.665,179.7264,1.7318,0.0000
C01536=95.882,-28.347,81.086,-179.9676,0.1107,0.0000
C01537=93.690,-34.955,81.363,-179.9953,0.0126,0.0000
C01538=90.965,-41.532,81.363,-179.9944,0.0123,0.0000
C01539=87.843,-47.755,81.086,-179.9446,0.1012,0.0000
C01540=83.804,-52.743,80.665,-178.5819,1.0314,0.0000
C01541=78.157,-54.900,80.245,-176.3975,0.3795,0.0000
C01542=72.072,-53.787,79.725,-174.8725,-2.5312,0.0000
C01543=66.340,-49.670,78.729,-175.2909,-3.4593,0.0000
C01544=60.266,-44.964,76.674,-175.7972,-3.0823,0.0000
C01545=54.746,-40.676,73.927,-176.5797,-2.4424,0.0000
C01546=50.430,-37.512,71.215,-178.6243,-0.9013,0.0000
C01547=47.226,-36.294,69.238,159.8058,-0.7740,0.0000
C01548=44.411,-37.931,68.453,153.5776,-22.3078,0.0000
C01549=42.621,-39.816,68.419,155.7180,-26.0884,0.0000
C01550=41.238,-41.238,68.442,154.7988,-25.2023,0.0000
C01551=39.816,-42.621,68.419,153.9110,-24.2815,0.0000
C01552=37.931,-44.412,68.453,157.6945,-26.4234,0.0000
C01553=36.294,-47.226,69.238,179.2264,-20.1937,0.0000
C01554=37.512,-50.430,71.215,179.0987,1.3757,0.0000
C01555=40.676,-54.746,73.927,177.5576,3.4203,0.0000
C01556=44.964,-60.266,76.674,176.9177,4.2028,0.0000
C01557=49.670,-66.340,78.729,176.5407,4.7091,0.0000
C01558=53.787,-72.072,79.725,177.4688,5.1275,0.0000
C01559=54.900,-78.157,80.245,-179.6205,3.6025,0.0000
C01560=52.743,-83.804,80.665,-178.9686,1.4181,0.0000
C01561=47.755,-87.843,81.086,-179.8988,0.0554,0.0000
C01562=41.532,-90.965,81.363,-179.9877,0.0056,0.0000
C01563=34.955,-93.690,81.363,-179.9874,0.0047,0.0000
C01564=28.347,-95.882,81.086,-179.8893,0.0324,0.0000
C01565=21.964,-96.553,80.665,-178.2682,-0.2736,0.0000
C01566=16.445,-94.085,80.245,-177.1832,-2.2811,0.0000
C01567=12.929,-88.996,79.725,-178.1562,-5.4103,0.0000
C01568=11.787,-82.032,78.729,-179.1118,-5.7669,0.0000
C01569=10.820,-74.409,76.674,-179.2045,-5.1449,0.0000
C01570=9.949,-67.473,73.927,-179.3067,-4.1423,0.0000
C01571=9.135,-62.185,71.215,-179.6644,-1.6099,0.0000
C01572=7.730,-59.058,69.238,164.9099,14.0649,0.0000
C01573=4.582,-58.225,68.453,147.3209,3.5043,0.0000
C01574=1.984,-58.291,68.419,146.3668,-1.5596,0.0000
C01575=0.000,-58.319,68.442,146.3550,-0.0009,0.0000
C01576=0.000,-58.319,68.442,146.3550,-0.0009,0.0000
C01577=-1.983,-58.291,68.419,146.3668,1.5606,0.0000
C01578=-4.583,-58.225,68.453,147.3217,-3.5071,0.0000
C01579=-7.730,-59.058,69.238,164.9105,-14.0648,0.0000
C01580=-9.135,-62.185,71.215,-179.6644,1.6099,0.0000
C01581=-9.949,-67.473,73.927,-179.3067,4.1423,0.0000
C01582=-10.820,-74.409,76.674,-179.2045,5.1449,0.0000
C01583=-11.787,-82.032,78.729,-179.1118,5.7669,0.0000
C01584=-12.929,-88.996,79.725,-178.1562,5.4103,0.0000
C01585=-16.445,-94.085,80.245,-177.1832,2.2811,0.0000
C01586=-21.964,-96.553,80.665,-178.2682,0.2736,0.0000
C01587=-28.347,-95.882,81.086,-179.8893,-0.0324,0.0000
C01588=-34.955,-93.690,81.363,-179.9874,-0.0047,0.0000
C01589=-41.532,-90.965,81.363,-179.9877,-0.0056,0.0000
C01590=-47.755,-87.843,81.086,-179.8988,-0.0554,0.0000
C01591=-52.743,-83.804,80.665,-178.9686,-1.4181,0.0000
C01592=-54.900,-78.157,80.245,-179.6205,-3.6025,0.0000
C01593=-53.787,-72.072,79.725,177.4688,-5.1275,0.0000
C01594=-49.670,-66.340,78.729,176.5407,-4.7091,0.0000
C01595=-44.964,-60.266,76.674,176.9177,-4.2028,0.0000
C01596=-40.676,-54.746,73.927,177.5576,-3.4203,0.0000
C01597=-37.512,-50.430,71.215,179.0987,-1.3757,0.0000
C01598=-36.294,-47.226,69.238,179.2260,20.1942,0.0000
C01599=-37.931,-44.411,68.453,157.6922,26.4224,0.0000
C01600=-39.816,-42.621,68.419,153.9116,24.2820,0.0000
C01601=-41.238,-41.238,68.442,154.7977,25.2012,0.0000
C01602=-42.621,-39.816,68.419,155.7185,26.0890,0.0000
C01603=-44.412,-37.931,68.453,153.5766,22.3055,0.0000
C01604=-47.226,-36.294,69.238,159.8063,0.7736,0.0000
C01605=-50.430,-37.512,71.215,-178.6243,0.9013,0.0000
C01606=-54.746,-40.676,73.927,-176.5797,2.4424,0.0000
C01607=-60.266,-44.964,76.674,-175.7972,3.0823,0.0000
C01608=-66.340,-49.670,78.729,-175.2909,3.4593,0.0000
C01609=-72.072,-53.787,79.725,-174.8725,2.5312,0.0000
C01610=-78.157,-54.900,80.245,-176.3975,-0.3795,0.0000
C01611=-83.804,-52.743,80.665,-178.5819,-1.0314,0.0000
C01612=-87.843,-47.755,81.086,-179.9446,-0.1012,0.0000
C01613=-90.965,-41.532,81.363,-179.9944,-0.0123,0.0000
C01614=-93.690,-34.955,81.363,-179.9953,-0.0126,0.0000
C01615=-95.882,-28.347,81.086,-179.9676,-0.1107,0.0000
C01616=-96.553,-21.964,80.665,179.7264,-1.7318,0.0000
C01617=-94.085,-16.445,80.245,177.7189,-2.8168,0.0000
C01618=-88.996,-12.929,79.725,174.5897,-1.8438,0.0000
C01619=-82.032,-11.787,78.729,174.2331,-0.8882,0.0000
C01620=-74.409,-10.820,76.674,174.8551,-0.7955,0.0000
C01621=-67.473,-9.949,73.927,175.8577,-0.6933,0.0000
C01622=-62.185,-9.135,71.215,178.3901,-0.3356,0.0000
C01623=-59.058,-7.730,69.238,-165.9351,15.0901,0.0000
C01624=-58.225,-4.582,68.453,-176.4957,32.6791,0.0000
C01625=-58.291,-1.984,68.419,178.4404,33.6332,0.0000
C01626=-58.319,0.000,68.442,179.9991,33.6450,0.0000
C01627=-58.291,1.983,68.419,-178.4394,33.6332,0.0000
C01628=-58.225,4.583,68.453,176.4929,32.6783,0.0000
C01629=-59.058,7.730,69.238,165.9352,15.0895,0.0000
C01630=-62.185,9.135,71.215,-178.3901,-0.3356,0.0000
C01631=-67.473,9.949,73.927,-175.8577,-0.6933,0.0000
C01632=-74.409,10.820,76.674,-174.8551,-0.7955,0.0000
C01633=-82.032,11.787,78.729,-174.2331,-0.8882,0.0000
C01634=-88.996,12.929,79.725,-174.5897,-1.8438,0.0000
C01635=-94.085,16.445,80.245,-177.7189,-2.8168,0.0000
C01636=-96.553,21.964,80.665,-179.7264,-1.7318,0.0000
C01637=-95.882,28.347,81.086,179.9676,-0.1107,0.0000
C01638=-93.690,34.955,81.363,179.9953,-0.0126,0.0000
C01639=-90.965,41.532,81.363,179.9944,-0.0123,0.0000
C01640=-87.843,47.755,81.086,179.9446,-0.1012,0.0000
C01641=-83.804,52.743,80.665,178.5819,-1.0314,0.0000
C01642=-78.157,54.900,80.245,176.3975,-0.3795,0.0000
C01643=-72.072,53.787,79.725,174.8725,2.5312,0.0000
C01644=-66.340,49.670,78.729,175.2909,3.4593,0.0000
C01645=-60.266,44.964,76.674,175.7972,3.0823,0.0000
C01646=-54.746,40.676,73.927,176.5797,2.4424,0.0000
C01647=-50.430,37.512,71.215,178.6243,0.9013,0.0000
C01648=-47.226,36.294,69.238,-159.8058,0.7740,0.0000
C01649=-44.411,37.931,68.453,-153.5776,22.3078,0.0000
C01650=-42.621,39.816,68.419,-155.7180,26.0884,0.0000
C01651=-41.238,41.238,68.442,-154.7988,25.2023,0.0000
C01652=-39.816,42.621,68.419,-153.9110,24.2815,0.0000
C01653=-37.931,44.412,68.453,-157.6945,26.4234,0.0000
C01654=-36.294,47.226,69.238,-179.2264,20.1937,0.0000
C01655=-37.512,50.430,71.215,-179.0987,-1.3757,0.0000
C01656=-40.676,54.746,73.927,-177.5576,-3.4203,0.0000
C01657=-44.964,60.266,76.674,-176.9177,-4.2028,0.0000
C01658=-49.670,66.340,78.729,-176.5407,-4.7091,0.0000
C01659=-53.787,72.072,79.725,-177.4688,-5.1275,0.0000
C01660=-54.900,78.157,80.245,179.6205,-3.6025,0.0000
C01661=-52.743,83.804,80.665,178.9686,-1.4181,0.0000
C01662=-47.755,87.843,81.086,179.8988,-0.0554,0.0000
C01663=-41.532,90.965,81.363,179.9877,-0.0056,0.0000
C01664=-34.955,93.690,81.363,179.9874,-0.0047,0.0000
C01665=-28.347,95.882,81.086,179.8893,-0.0324,0.0000
C01666=-21.964,96.553,80.665,178.2682,0.2736,0.0000
C01667=-16.445,94.085,80.245,177.1832,2.2811,0.0000
C01668=-12.929,88.996,79.725,178.1562,5.4103,0.0000
C01669=-11.787,82.032,78.729,179.1118,5.7669,0.0000
C01670=-10.820,74.409,76.674,179.2045,5.1449,0.0000
C01671=-9.949,67.473,73.927,179.3067,4.1423,0.0000
C01672=-9.135,62.185,71.215,179.6644,1.6099,0.0000
C01673=-7.730,59.058,69.238,-164.9105,-14.0648,0.0000
C01674=-4.583,58.225,68.453,-147.3217,-3.5071,0.0000
C01675=-1.983,58.291,68.419,-146.3668,1.5606,0.0000
C01676=0.000,58.319,68.442,-146.3550,-0.0009,0.0000
C01677=0.000,57.118,70.285,-147.5034,-0.0009,0.0000
C01678=1.874,57.094,70.261,-147.5130,-1.4410,0.0000
C01679=4.398,57.039,70.297,-148.5403,3.6784,0.0000
C01680=7.507,57.930,71.114,-166.2856,13.3384,0.0000
C01681=8.875,61.204,73.167,179.6344,-1.8648,0.0000
C01682=9.674,66.709,75.971,179.3569,-3.9987,0.0000
C01683=10.553,73.885,78.794,179.2847,-4.7758,0.0000
C01684=11.527,81.722,80.892,179.2219,-5.2319,0.0000
C01685=12.662,88.851,81.904,178.3832,-4.8674,0.0000
C01686=16.202,94.056,82.431,177.4937,-2.0609,0.0000
C01687=21.776,96.587,82.857,178.4589,-0.2498,0.0000
C01688=28.231,95.920,83.283,179.9016,0.0287,0.0000
C01689=34.916,93.705,83.562,179.9888,0.0041,0.0000
C01690=41.570,90.949,83.562,179.9892,0.0050,0.0000
C01691=47.863,87.788,83.283,179.9101,0.0492,0.0000
C01692=52.900,83.695,82.857,179.0867,1.2664,0.0000
C01693=55.051,77.964,82.431,179.6845,3.2279,0.0000
C01694=53.873,71.781,81.904,-177.6947,4.5839,0.0000
C01695=49.635,65.937,80.892,-176.8436,4.2522,0.0000
C01696=44.783,59.707,78.794,-177.1234,3.8847,0.0000
C01697=40.330,54.011,75.971,-177.6240,3.2832,0.0000
C01698=37.003,49.553,73.167,-178.9395,1.5772,0.0000
C01699=35.654,46.271,71.114,-179.7188,-18.7891,0.0000
C01700=37.223,43.442,70.297,-158.8350,-25.5520,0.0000
C01701=39.047,41.697,70.261,-154.9186,-23.3867,0.0000
C01702=40.388,40.388,70.285,-155.7518,-24.2471,0.0000
C01703=41.696,39.047,70.261,-156.6139,-25.0820,0.0000
C01704=43.443,37.223,70.297,-154.4471,-21.1627,0.0000
C01705=46.271,35.654,71.114,-161.2114,-0.2808,0.0000
C01706=49.553,37.003,73.167,178.4228,-1.0605,0.0000
C01707=54.011,40.330,75.971,176.7168,-2.3760,0.0000
C01708=59.707,44.783,78.794,176.1153,-2.8766,0.0000
C01709=65.937,49.635,80.892,175.7478,-3.1564,0.0000
C01710=71.781,53.873,81.904,175.4161,-2.3053,0.0000
C01711=77.964,55.051,82.431,176.7721,0.3155,0.0000
C01712=83.695,52.900,82.857,178.7336,0.9133,0.0000
C01713=87.788,47.863,83.283,179.9508,0.0899,0.0000
C01714=90.949,41.570,83.562,179.9950,0.0108,0.0000
C01715=93.705,34.916,83.562,179.9959,0.0112,0.0000
C01716=95.920,28.231,83.283,179.9713,0.0984,0.0000
C01717=96.587,21.776,82.857,-179.7502,1.5411,0.0000
C01718=94.056,16.202,82.431,-177.9391,2.5063,0.0000
C01719=88.851,12.662,81.904,-175.1326,1.6168,0.0000
C01720=81.722,11.527,80.892,-174.7681,0.7781,0.0000
C01721=73.885,10.553,78.794,-175.2242,0.7153,0.0000
C01722=66.709,9.674,75.971,-176.0013,0.6431,0.0000
C01723=61.204,8.875,73.167,-178.1352,0.3656,0.0000
C01724=57.930,7.507,71.114,166.6616,-13.7144,0.0000
C01725=57.039,4.398,70.297,176.3216,-31.4597,0.0000
C01726=57.094,1.874,70.261,-178.5590,-32.4870,0.0000
C01727=57.118,0.000,70.285,-179.9991,-32.4966,0.0000
C01728=57.094,-1.874,70.261,178.5580,-32.4870,0.0000
C01729=57.039,-4.398,70.297,-176.3189,-31.4589,0.0000
C01730=57.930,-7.507,71.114,-166.6617,-13.7137,0.0000
C01731=61.204,-8.875,73.167,178.1352,0.3656,0.0000
C01732=66.709,-9.674,75.971,176.0013,0.6431,0.0000
C01733=73.885,-10.553,78.794,175.2242,0.7153,0.0000
C01734=81.722,-11.527,80.892,174.7681,0.7781,0.0000
C01735=88.851,-12.662,81.904,175.1326,1.6168,0.0000
C01736=94.056,-16.202,82.431,177.9391,2.5063,0.0000
C01737=96.587,-21.776,82.857,179.7502,1.5411,0.0000
C01738=95.920,-28.231,83.283,-179.9713,0.0984,0.0000
C01739=93.705,-34.916,83.562,-179.9959,0.0112,0.0000
C01740=90.949,-41.570,83.562,-179.9950,0.0108,0.0000
C01741=87.788,-47.863,83.283,-179.9508,0.0899,0.0000
C01742=83.695,-52.900,82.857,-178.7336,0.9133,0.0000
C01743=77.964,-55.051,82.431,-176.7721,0.3155,0.0000
C01744=71.781,-53.873,81.904,-175.4161,-2.3053,0.0000
C01745=65.937,-49.635,80.892,-175.7478,-3.1564,0.0000
C01746=59.707,-44.783,78.794,-176.1153,-2.8766,0.0000
C01747=54.011,-40.330,75.971,-176.7168,-2.3760,0.0000
C01748=49.553,-37.003,73.167,-178.4228,-1.0605,0.0000
C01749=46.271,-35.654,71.114,161.2109,-0.2812,0.0000
C01750=43.442,-37.223,70.297,154.4480,-21.1650,0.0000
C01751=41.697,-39.047,70.261,156.6133,-25.0814,0.0000
C01752=40.388,-40.388,70.285,155.7529,-24.2482,0.0000
C01753=39.047,-41.696,70.261,154.9180,-23.3861,0.0000
C01754=37.223,-43.443,70.297,158.8373,-25.5529,0.0000
C01755=35.654,-46.271,71.114,179.7192,-18.7886,0.0000
C01756=37.003,-49.553,73.167,178.9395,1.5772,0.0000
C01757=40.330,-54.011,75.971,177.6240,3.2832,0.0000
C01758=44.783,-59.707,78.794,177.1234,3.8847,0.0000
C01759=49.635,-65.937,80.892,176.8436,4.2522,0.0000
C01760=53.873,-71.781,81.904,177.6947,4.5839,0.0000
C01761=55.051,-77.964,82.431,-179.6845,3.2279,0.0000
C01762=52.900,-83.695,82.857,-179.0867,1.2664,0.0000
C01763=47.863,-87.788,83.283,-179.9101,0.0492,0.0000
C01764=41.570,-90.949,83.562,-179.9892,0.0050,0.0000
C01765=34.916,-93.705,83.562,-179.9888,0.0041,0.0000
C01766=28.231,-95.920,83.283,-179.9016,0.0287,0.0000
C01767=21.776,-96.587,82.857,-178.4589,-0.2498,0.0000
C01768=16.202,-94.056,82.431,-177.4937,-2.0609,0.0000
C01769=12.662,-88.851,81.904,-178.3832,-4.8674,0.0000
C01770=11.527,-81.722,80.892,-179.2219,-5.2319,0.0000
C01771=10.553,-73.885,78.794,-179.2847,-4.7758,0.0000
C01772=9.674,-66.709,75.971,-179.3569,-3.9987,0.0000
C01773=8.875,-61.204,73.167,-179.6344,-1.8648,0.0000
C01774=7.507,-57.930,71.114,166.2856,13.3384,0.0000
C01775=4.398,-57.039,70.297,148.5403,3.6784,0.0000
C01776=1.874,-57.094,70.261,147.5130,-1.4410,0.0000
C01777=0.000,-57.118,70.285,147.5034,-0.0009,0.0000
C01778=0.000,-57.118,70.285,147.5034,-0.0009,0.0000
C01779=-1.874,-57.094,70.261,147.5130,1.4420,0.0000
C01780=-4.398,-57.039,70.297,148.5411,-3.6811,0.0000
C01781=-7.507,-57.930,71.114,166.2863,-13.3383,0.0000
C01782=-8.875,-61.204,73.167,-179.6344,1.8648,0.0000
C01783=-9.674,-66.709,75.971,-179.3569,3.9987,0.0000
C01784=-10.553,-73.885,78.794,-179.2847,4.7758,0.0000
C01785=-11.527,-81.722,80.892,-179.2219,5.2319,0.0000
C01786=-12.662,-88.851,81.904,-178.3832,4.8674,0.0000
C01787=-16.202,-94.056,82.431,-177.4937,2.0609,0.0000
C01788=-21.776,-96.587,82.857,-178.4589,0.2498,0.0000
C01789=-28.231,-95.920,83.283,-179.9016,-0.0287,0.0000
C01790=-34.916,-93.705,83.562,-179.9888,-0.0041,0.0000
C01791=-41.570,-90.949,83.562,-179.9892,-0.0050,0.0000
C01792=-47.863,-87.788,83.283,-179.9101,-0.0492,0.0000
C01793=-52.900,-83.695,82.857,-179.0867,-1.2664,0.0000
C01794=-55.051,-77.964,82.431,-179.6845,-3.2279,0.0000
C01795=-53.873,-71.781,81.904,177.6947,-4.5839,0.0000
C01796=-49.635,-65.937,80.892,176.8436,-4.2522,0.0000
C01797=-44.783,-59.707,78.794,177.1234,-3.8847,0.0000
C01798=-40.330,-54.011,75.971,177.6240,-3.2832,0.0000
C01799=-37.003,-49.553,73.167,178.9395,-1.5772,0.0000
C01800=-35.654,-46.271,71.114,179.7188,18.7891,0.0000
C01801=-37.223,-43.442,70.297,158.8350,25.5520,0.0000
C01802=-39.047,-41.697,70.261,154.9186,23.3867,0.0000
C01803=-40.388,-40.388,70.285,155.7518,24.2471,0.0000
C01804=-41.696,-39.047,70.261,156.6139,25.0820,0.0000
C01805=-43.443,-37.223,70.297,154.4471,21.1627,0.0000
C01806=-46.271,-35.654,71.114,161.2114,0.2808,0.0000
C01807=-49.553,-37.003,73.167,-178.4228,1.0605,0.0000
C01808=-54.011,-40.330,75.971,-176.7168,2.3760,0.0000
C01809=-59.707,-44.783,78.794,-176.1153,2.8766,0.0000
C01810=-65.937,-49.635,80.892,-175.7478,3.1564,0.0000
C01811=-71.781,-53.873,81.904,-175.4161,2.3053,0.0000
C01812=-77.964,-55.051,82.431,-176.7721,-0.3155,0.0000
C01813=-83.695,-52.900,82.857,-178.7336,-0.9133,0.0000
C01814=-87.788,-47.863,83.283,-179.9508,-0.0899,0.0000
C01815=-90.949,-41.570,83.562,-179.9950,-0.0108,0.0000
C01816=-93.705,-34.916,83.562,-179.9959,-0.0112,0.0000
C01817=-95.920,-28.231,83.283,-179.9713,-0.0984,0.0000
C01818=-96.587,-21.776,82.857,179.7502,-1.5411,0.0000
C01819=-94.056,-16.202,82.431,177.9391,-2.5063,0.0000
C01820=-88.851,-12.662,81.904,175.1326,-1.6168,0.0000
C01821=-81.722,-11.527,80.892,174.7681,-0.7781,0.0000
C01822=-73.885,-10.553,78.794,175.2242,-0.7153,0.0000
C01823=-66.709,-9.674,75.971,176.0013,-0.6431,0.0000
C01824=-61.204,-8.875,73.167,178.1352,-0.3656,0.0000
C01825=-57.930,-7.507,71.114,-166.6616,13.7144,0.0000
C01826=-57.039,-4.398,70.297,-176.3216,31.4597,0.0000
C01827=-57.094,-1.874,70.261,178.5590,32.4870,0.0000
C01828=-57.118,0.000,70.285,179.9991,32.4966,0.0000
C01829=-57.094,1.874,70.261,-178.5580,32.4870,0.0000
C01830=-57.039,4.398,70.297,176.3189,31.4589,0.0000
C01831=-57.930,7.507,71.114,166.6617,13.7137,0.0000
C01832=-61.204,8.875,73.167,-178.1352,-0.3656,0.0000
C01833=-66.709,9.674,75.971,-176.0013,-0.6431,0.0000
C01834=-73.885,10.553,78.794,-175.2242,-0.7153,0.0000
C01835=-81.722,11.527,80.892,-174.7681,-0.7781,0.0000
C01836=-88.851,12.662,81.904,-175.1326,-1.6168,0.0000
C01837=-94.056,16.202,82.431,-177.9391,-2.5063,0.0000
C01838=-96.587,21.776,82.857,-179.7502,-1.5411,0.0000
C01839=-95.920,28.231,83.283,179.9713,-0.0984,0.0000
C01840=-93.705,34.916,83.562,179.9959,-0.0112,0.0000
C01841=-90.949,41.570,83.562,179.9950,-0.0108,0.0000
C01842=-87.788,47.863,83.283,179.9508,-0.0899,0.0000
C01843=-83.695,52.900,82.857,178.7336,-0.9133,0.0000
C01844=-77.964,55.051,82.431,176.7721,-0.3155,0.0000
C01845=-71.781,53.873,81.904,175.4161,2.3053,0.0000
C01846=-65.937,49.635,80.892,175.7478,3.1564,0.0000
C01847=-59.707,44.783,78.794,176.1153,2.8766,0.0000
C01848=-54.011,40.330,75.971,176.7168,2.3760,0.0000
C01849=-49.553,37.003,73.167,178.4228,1.0605,0.0000
C01850=-46.271,35.654,71.114,-161.2109,0.2812,0.0000
C01851=-43.442,37.223,70.297,-154.4480,21.1650,0.0000
C01852=-41.697,39.047,70.261,-156.6133,25.0814,0.0000
C01853=-40.388,40.388,70.285,-155.7529,24.2482,0.0000
C01854=-39.047,41.696,70.261,-154.9180,23.3861,0.0000
C01855=-37.223,43.443,70.297,-158.8373,25.5529,0.0000
C01856=-35.654,46.271,71.114,-179.7192,18.7886,0.0000
C01857=-37.003,49.553,73.167,-178.9395,-1.5772,0.0000
C01858=-40.330,54.011,75.971,-177.6240,-3.2832,0.0000
C01859=-44.783,59.707,78.794,-177.1234,-3.8847,0.0000
C01860=-49.635,65.937,80.892,-176.8436,-4.2522,0.0000
C01861=-53.873,71.781,81.904,-177.6947,-4.5839,0.0000
C01862=-55.051,77.964,82.431,179.6845,-3.2279,0.0000
C01863=-52.900,83.695,82.857,179.0867,-1.2664,0.0000
C01864=-47.863,87.788,83.283,179.9101,-0.0492,0.0000
C01865=-41.570,90.949,83.562,179.9892,-0.0050,0.0000
C01866=-34.916,93.705,83.562,179.9888,-0.0041,0.0000
C01867=-28.231,95.920,83.283,179.9016,-0.0287,0.0000
C01868=-21.776,96.587,82.857,178.4589,0.2498,0.0000
C01869=-16.202,94.056,82.431,177.4937,2.0609,0.0000
C01870=-12.662,88.851,81.904,178.3832,4.8674,0.0000
C01871=-11.527,81.722,80.892,179.2219,5.2319,0.0000
C01872=-10.553,73.885,78.794,179.2847,4.7758,0.0000
C01873=-9.674,66.709,75.971,179.3569,3.9987,0.0000
C01874=-8.875,61.204,73.167,179.6344,1.8648,0.0000
C01875=-7.507,57.930,71.114,-166.2863,-13.3383,0.0000
C01876=-4.398,57.039,70.297,-148.5411,-3.6811,0.0000
C01877=-1.874,57.094,70.261,-147.5130,1.4420,0.0000
